LIN {X 0,Y 334.932,Z 502.73,A -85,B 0,C 180,E1 -14665.187,E2 -14665.187} C_VEL
LIN {X 0,Y 334.415,Z 506.51,A -85,B 0,C 180,E1 -14666.99,E2 -14666.99} C_VEL
LIN {X 0,Y 334.012,Z 509.299,A -85,B 0,C 180,E1 -14668.796,E2 -14668.796} C_VEL
LIN {X 0,Y 333.863,Z 511.532,A -85,B 0,C 180,E1 -14671.207,E2 -14671.207} C_VEL
LIN {X 0,Y 333.779,Z 512.102,A -85,B 0,C 180,E1 -14672.415,E2 -14672.415} C_VEL
LIN {X 0,Y 333.646,Z 512.277,A -85,B 0,C 180,E1 -14673.624,E2 -14673.624} C_VEL
LIN {X 0,Y 334.045,Z 511.395,A -85,B 0,C 180,E1 -14676.04,E2 -14676.04} C_VEL
LIN {X 0,Y 334.412,Z 510.379,A -85,B 0,C 180,E1 -14677.245,E2 -14677.245} C_VEL
LIN {X 0,Y 334.959,Z 507.296,A -85,B 0,C 180,E1 -14679.548,E2 -14679.548} C_VEL
LIN {X 0,Y 335.704,Z 503.489,A -85,B 0,C 180,E1 -14681.473,E2 -14681.473} C_VEL
LIN {X 0,Y 336.395,Z 498.792,A -85,B 0,C 180,E1 -14683.287,E2 -14683.287} C_VEL
LIN {X 0,Y 337.32,Z 492.834,A -85,B 0,C 180,E1 -14685.097,E2 -14685.097} C_VEL
LIN {X 0,Y 338.463,Z 485.332,A -85,B 0,C 180,E1 -14686.901,E2 -14686.901} C_VEL
LIN {X 0,Y 339.867,Z 475.902,A -85,B 0,C 180,E1 -14688.695,E2 -14688.695} C_VEL
LIN {X 0,Y 341.064,Z 466.087,A -85,B 0,C 180,E1 -14690.192,E2 -14690.192} C_VEL
LIN {X 0,Y 342.197,Z 454.989,A -85,B 0,C 180,E1 -14691.539,E2 -14691.539} C_VEL
LIN {X 0,Y 343.141,Z 443.458,A -85,B 0,C 180,E1 -14692.639,E2 -14692.639} C_VEL
LIN {X 0,Y 343.723,Z 434.102,A -85,B 0,C 180,E1 -14693.339,E2 -14693.339} C_VEL
LIN {X 0,Y 339.861,Z 422.675,A -85,B 0,C 180,E1 -14694.326,E2 -14694.326} C_VEL
LIN {X 0,Y 334.962,Z 410.747,A -85,B 0,C 180,E1 -14695.19,E2 -14695.19} C_VEL
LIN {X 0,Y 333.811,Z 407.943,A -85,B 0,C 180,E1 -14695.364,E2 -14695.364} C_VEL
LIN {X 0,Y 333.742,Z 407.533,A -85,B 0,C 180,E1 -14695.441,E2 -14695.441} C_VEL
LIN {X 0,Y 333.717,Z 407.543,A -85,B 0,C 180,E1 -14698.973,E2 -14698.973} C_VEL
LIN {X 0,Y 333.649,Z 407.552,A -85,B 0,C 180,E1 -14702.587,E2 -14702.587} C_VEL
LIN {X 0,Y 333.682,Z 407.549,A -85,B 0,C 180,E1 -14706.139,E2 -14706.139} C_VEL
LIN {X 0,Y 333.652,Z 407.539,A -85,B 0,C 180,E1 -14709.193,E2 -14709.193} C_VEL
LIN {X 0,Y 333.638,Z 407.548,A -85,B 0,C 180,E1 -14712.5,E2 -14712.5} C_VEL
LIN {X 0,Y 333.591,Z 407.549,A -85,B 0,C 180,E1 -14716.485,E2 -14716.485} C_VEL
LIN {X 0,Y 333.654,Z 407.539,A -85,B 0,C 180,E1 -14719.315,E2 -14719.315} C_VEL
LIN {X 0,Y 333.642,Z 407.519,A -85,B 0,C 180,E1 -14721.721,E2 -14721.721} C_VEL
LIN {X 0,Y 332.986,Z 407.614,A -85,B 0,C 180,E1 -14722.729,E2 -14722.729} C_VEL
LIN {X 0,Y 330.166,Z 407.982,A -85,B 0,C 180,E1 -14724.369,E2 -14724.369} C_VEL
LIN {X 0,Y 327.763,Z 408.288,A -85,B 0,C 180,E1 -14725.697,E2 -14725.697} C_VEL
LIN {X 0,Y 326.717,Z 408.412,A -85,B 0,C 180,E1 -14726.725,E2 -14726.725} C_VEL
LIN {X 0,Y 326.623,Z 408.419,A -85,B 0,C 180,E1 -14727.073,E2 -14727.073} C_VEL
LIN {X 0,Y 326.653,Z 408.377,A -85,B 0,C 180,E1 -14730.34,E2 -14730.34} C_VEL
LIN {X 0,Y 326.695,Z 408.413,A -85,B 0,C 180,E1 -14734.516,E2 -14734.516} C_VEL
LIN {X 0,Y 326.643,Z 408.545,A -85,B 0,C 180,E1 -14737.811,E2 -14737.811} C_VEL
LIN {X 0,Y 330.893,Z 422.806,A -85,B 0,C 180,E1 -14739.156,E2 -14739.156} C_VEL
LIN {X 0,Y 333.894,Z 433.415,A -85,B 0,C 180,E1 -14740.319,E2 -14740.319} C_VEL
LIN {X 0,Y 332.75,Z 446.544,A -85,B 0,C 180,E1 -14741.759,E2 -14741.759} C_VEL
LIN {X 0,Y 331.562,Z 458.658,A -85,B 0,C 180,E1 -14743.372,E2 -14743.372} C_VEL
LIN {X 0,Y 330.264,Z 470.023,A -85,B 0,C 180,E1 -14745.205,E2 -14745.205} C_VEL
LIN {X 0,Y 329.393,Z 479.499,A -85,B 0,C 180,E1 -14747.054,E2 -14747.054} C_VEL
LIN {X 0,Y 328.405,Z 488.672,A -85,B 0,C 180,E1 -14749.207,E2 -14749.207} C_VEL
LIN {X 0,Y 327.734,Z 496.151,A -85,B 0,C 180,E1 -14751.366,E2 -14751.366} C_VEL
LIN {X 0,Y 327.381,Z 501.397,A -85,B 0,C 180,E1 -14753.219,E2 -14753.219} C_VEL
LIN {X 0,Y 326.834,Z 505.753,A -85,B 0,C 180,E1 -14755.065,E2 -14755.065} C_VEL
LIN {X 0,Y 326.643,Z 508.141,A -85,B 0,C 180,E1 -14756.299,E2 -14756.299} C_VEL
LIN {X 0,Y 326.854,Z 511.779,A -85,B 0,C 180,E1 -14758.768,E2 -14758.768} C_VEL
LIN {X 0,Y 326.937,Z 514.089,A -85,B 0,C 180,E1 -14761.231,E2 -14761.231} C_VEL
LIN {X 0,Y 327.345,Z 515.047,A -85,B 0,C 180,E1 -14763.693,E2 -14763.693} C_VEL
LIN {X 0,Y 327.978,Z 514.689,A -85,B 0,C 180,E1 -14766.15,E2 -14766.15} C_VEL
LIN {X 0,Y 328.936,Z 512.991,A -85,B 0,C 180,E1 -14768.601,E2 -14768.601} C_VEL
LIN {X 0,Y 330.253,Z 509.9,A -85,B 0,C 180,E1 -14771.042,E2 -14771.042} C_VEL
LIN {X 0,Y 331.845,Z 505.402,A -85,B 0,C 180,E1 -14773.471,E2 -14773.471} C_VEL
LIN {X 0,Y 333.337,Z 501.026,A -85,B 0,C 180,E1 -14775.28,E2 -14775.28} C_VEL
LIN {X 0,Y 335.699,Z 493.646,A -85,B 0,C 180,E1 -14777.672,E2 -14777.672} C_VEL
LIN {X 0,Y 338.143,Z 485.587,A -85,B 0,C 180,E1 -14779.739,E2 -14779.739} C_VEL
LIN {X 0,Y 340.863,Z 475.682,A -85,B 0,C 180,E1 -14781.785,E2 -14781.785} C_VEL
LIN {X 0,Y 343.444,Z 465.427,A -85,B 0,C 180,E1 -14783.518,E2 -14783.518} C_VEL
LIN {X 0,Y 346.007,Z 454.2,A -85,B 0,C 180,E1 -14785.088,E2 -14785.088} C_VEL
LIN {X 0,Y 346.695,Z 451.167,A -85,B 0,C 180,E1 -14785.448,E2 -14785.448} C_VEL
LIN {X 0,Y 346.751,Z 449.531,A -85,B 0,C 180,E1 -14785.698,E2 -14785.698} C_VEL
LIN {X 0,Y 344.955,Z 442.595,A -85,B 0,C 180,E1 -14787.072,E2 -14787.072} C_VEL
LIN {X 0,Y 342.423,Z 435.536,A -85,B 0,C 180,E1 -14788.594,E2 -14788.594} C_VEL
LIN {X 0,Y 338.778,Z 427.656,A -85,B 0,C 180,E1 -14790.489,E2 -14790.489} C_VEL
LIN {X 0,Y 336.804,Z 424.314,A -85,B 0,C 180,E1 -14791.444,E2 -14791.444} C_VEL
LIN {X 0,Y 334.026,Z 421.028,A -85,B 0,C 180,E1 -14792.688,E2 -14792.688} C_VEL
LIN {X 0,Y 331.005,Z 418.156,A -85,B 0,C 180,E1 -14794.099,E2 -14794.099} C_VEL
LIN {X 0,Y 328.685,Z 416.422,A -85,B 0,C 180,E1 -14795.262,E2 -14795.262} C_VEL
LIN {X 0,Y 328.179,Z 415.479,A -85,B 0,C 180,E1 -14795.701,E2 -14795.701} C_VEL
LIN {X 0,Y 328.67,Z 417.798,A -85,B 0,C 180,E1 -14798.324,E2 -14798.324} C_VEL
LIN {X 0,Y 329.451,Z 421.54,A -85,B 0,C 180,E1 -14801.699,E2 -14801.699} C_VEL
LIN {X 0,Y 330.309,Z 425.475,A -85,B 0,C 180,E1 -14804.599,E2 -14804.599} C_VEL
LIN {X 0,Y 331.337,Z 430.877,A -85,B 0,C 180,E1 -14807.935,E2 -14807.935} C_VEL
LIN {X 0,Y 331.487,Z 434.338,A -85,B 0,C 180,E1 -14809.752,E2 -14809.752} C_VEL
LIN {X 0,Y 329.383,Z 444.47,A -85,B 0,C 180,E1 -14814.174,E2 -14814.174} C_VEL
LIN {X 0,Y 329.004,Z 447.721,A -85,B 0,C 180,E1 -14815.43,E2 -14815.43} C_VEL
LIN {X 0,Y 330.074,Z 452.747,A -85,B 0,C 180,E1 -14816.199,E2 -14816.199} C_VEL
LIN {X 0,Y 331.177,Z 456.012,A -85,B 0,C 180,E1 -14816.784,E2 -14816.784} C_VEL
LIN {X 0,Y 332.291,Z 460.774,A -85,B 0,C 180,E1 -14817.472,E2 -14817.472} C_VEL
LIN {X 0,Y 333.055,Z 464.005,A -85,B 0,C 180,E1 -14817.942,E2 -14817.942} C_VEL
LIN {X 0,Y 334.284,Z 469.371,A -85,B 0,C 180,E1 -14818.683,E2 -14818.683} C_VEL
LIN {X 0,Y 336.767,Z 483.631,A -85,B 0,C 180,E1 -14820.487,E2 -14820.487} C_VEL
LIN {X 0,Y 338.023,Z 497.366,A -85,B 0,C 180,E1 -14822.075,E2 -14822.075} C_VEL
LIN {X 0,Y 338.104,Z 510.892,A -85,B 0,C 180,E1 -14823.59,E2 -14823.59} C_VEL
LIN {X 0,Y 336.94,Z 523.468,A -85,B 0,C 180,E1 -14825.014,E2 -14825.014} C_VEL
LIN {X 0,Y 335.439,Z 536.699,A -85,B 0,C 180,E1 -14826.704,E2 -14826.704} C_VEL
LIN {X 0,Y 332.995,Z 548.466,A -85,B 0,C 180,E1 -14828.356,E2 -14828.356} C_VEL
LIN {X 0,Y 330.787,Z 559.176,A -85,B 0,C 180,E1 -14830.126,E2 -14830.126} C_VEL
LIN {X 0,Y 328.676,Z 570.047,A -85,B 0,C 180,E1 -14832.258,E2 -14832.258} C_VEL
LIN {X 0,Y 327.218,Z 579.19,A -85,B 0,C 180,E1 -14834.425,E2 -14834.425} C_VEL
LIN {X 0,Y 326.321,Z 585.851,A -85,B 0,C 180,E1 -14836.295,E2 -14836.295} C_VEL
LIN {X 0,Y 325.733,Z 593.228,A -85,B 0,C 180,E1 -14838.802,E2 -14838.802} C_VEL
LIN {X 0,Y 325.614,Z 598.959,A -85,B 0,C 180,E1 -14841.309,E2 -14841.309} C_VEL
LIN {X 0,Y 325.829,Z 603.168,A -85,B 0,C 180,E1 -14843.807,E2 -14843.807} C_VEL
LIN {X 0,Y 326.041,Z 604.717,A -85,B 0,C 180,E1 -14845.052,E2 -14845.052} C_VEL
LIN {X 0,Y 326.172,Z 605.881,A -85,B 0,C 180,E1 -14846.292,E2 -14846.292} C_VEL
LIN {X 0,Y 326.574,Z 607.099,A -85,B 0,C 180,E1 -14848.766,E2 -14848.766} C_VEL
LIN {X 0,Y 326.764,Z 607.138,A -85,B 0,C 180,E1 -14849.999,E2 -14849.999} C_VEL
LIN {X 0,Y 326.616,Z 606.741,A -85,B 0,C 180,E1 -14851.232,E2 -14851.232} C_VEL
LIN {X 0,Y 326.459,Z 605.959,A -85,B 0,C 180,E1 -14852.466,E2 -14852.466} C_VEL
LIN {X 0,Y 326.23,Z 603.225,A -85,B 0,C 180,E1 -14854.942,E2 -14854.942} C_VEL
LIN {X 0,Y 326.053,Z 599.629,A -85,B 0,C 180,E1 -14857.027,E2 -14857.027} C_VEL
LIN {X 0,Y 325.922,Z 594.313,A -85,B 0,C 180,E1 -14859.306,E2 -14859.306} C_VEL
LIN {X 0,Y 326.074,Z 587.723,A -85,B 0,C 180,E1 -14861.499,E2 -14861.499} C_VEL
LIN {X 0,Y 326.518,Z 579.433,A -85,B 0,C 180,E1 -14863.694,E2 -14863.694} C_VEL
LIN {X 0,Y 327.31,Z 570.812,A -85,B 0,C 180,E1 -14865.568,E2 -14865.568} C_VEL
LIN {X 0,Y 328.372,Z 560.421,A -85,B 0,C 180,E1 -14867.434,E2 -14867.434} C_VEL
LIN {X 0,Y 329.62,Z 550.112,A -85,B 0,C 180,E1 -14868.973,E2 -14868.973} C_VEL
LIN {X 0,Y 331.041,Z 537.717,A -85,B 0,C 180,E1 -14870.504,E2 -14870.504} C_VEL
LIN {X 0,Y 331.642,Z 529.973,A -85,B 0,C 180,E1 -14871.322,E2 -14871.322} C_VEL
LIN {X 0,Y 330.688,Z 516.048,A -85,B 0,C 180,E1 -14872.603,E2 -14872.603} C_VEL
LIN {X 0,Y 329.222,Z 500.525,A -85,B 0,C 180,E1 -14873.76,E2 -14873.76} C_VEL
LIN {X 0,Y 327.764,Z 485.333,A -85,B 0,C 180,E1 -14874.63,E2 -14874.63} C_VEL
LIN {X 0,Y 326.846,Z 476.144,A -85,B 0,C 180,E1 -14875.043,E2 -14875.043} C_VEL
LIN {X 0,Y 327.719,Z 465.495,A -85,B 0,C 180,E1 -14878.914,E2 -14878.914} C_VEL
LIN {X 0,Y 328.904,Z 454.506,A -85,B 0,C 180,E1 -14882.961,E2 -14882.961} C_VEL
LIN {X 0,Y 330.094,Z 444.79,A -85,B 0,C 180,E1 -14886.592,E2 -14886.592} C_VEL
LIN {X 0,Y 331.502,Z 435.163,A -85,B 0,C 180,E1 -14890.251,E2 -14890.251} C_VEL
LIN {X 0,Y 331.337,Z 431.895,A -85,B 0,C 180,E1 -14891.564,E2 -14891.564} C_VEL
LIN {X 0,Y 329.548,Z 423.114,A -85,B 0,C 180,E1 -14895.27,E2 -14895.27} C_VEL
LIN {X 0,Y 327.775,Z 414.147,A -85,B 0,C 180,E1 -14899.251,E2 -14899.251} C_VEL
LIN {X 0,Y 326.642,Z 408.424,A -85,B 0,C 180,E1 -14901.952,E2 -14901.952} C_VEL
LIN {X 0,Y 326.598,Z 408.425,A -85,B 0,C 180,E1 -14905.98,E2 -14905.98} C_VEL
LIN {X 0,Y 326.651,Z 408.417,A -85,B 0,C 180,E1 -14910.34,E2 -14910.34} C_VEL
LIN {X 0,Y 326.68,Z 408.415,A -85,B 0,C 180,E1 -14914.516,E2 -14914.516} C_VEL
LIN {X 0,Y 326.636,Z 408.421,A -85,B 0,C 180,E1 -14918.545,E2 -14918.545} C_VEL
LIN {X 0,Y 326.734,Z 408.412,A -85,B 0,C 180,E1 -14921.177,E2 -14921.177} C_VEL
LIN {X 0,Y 326.753,Z 408.407,A -85,B 0,C 180,E1 -14925.433,E2 -14925.433} C_VEL
LIN {X 0,Y 326.763,Z 408.408,A -85,B 0,C 180,E1 -14928.839,E2 -14928.839} C_VEL
LIN {X 0,Y 326.969,Z 408.381,A -85,B 0,C 180,E1 -14932.59,E2 -14932.59} C_VEL
LIN {X 0,Y 326.77,Z 408.406,A -85,B 0,C 180,E1 -14935.065,E2 -14935.065} C_VEL
LIN {X 0,Y 327.059,Z 408.368,A -85,B 0,C 180,E1 -14937.537,E2 -14937.537} C_VEL
LIN {X 0,Y 327.208,Z 408.348,A -85,B 0,C 180,E1 -14940,E2 -14940} C_VEL
LIN {X 0,Y 327.059,Z 408.369,A -85,B 0,C 180,E1 -14942.463,E2 -14942.463} C_VEL
LIN {X 0,Y 326.961,Z 408.375,A -85,B 0,C 180,E1 -14946.673,E2 -14946.673} C_VEL
LIN {X 0,Y 326.806,Z 408.393,A -85,B 0,C 180,E1 -14949.907,E2 -14949.907} C_VEL
LIN {X 0,Y 326.751,Z 408.406,A -85,B 0,C 180,E1 -14953.686,E2 -14953.686} C_VEL
LIN {X 0,Y 326.69,Z 408.412,A -85,B 0,C 180,E1 -14957.529,E2 -14957.529} C_VEL
LIN {X 0,Y 326.656,Z 408.418,A -85,B 0,C 180,E1 -14960.136,E2 -14960.136} C_VEL
LIN {X 0,Y 326.643,Z 408.42,A -85,B 0,C 180,E1 -14964.13,E2 -14964.13} C_VEL
LIN {X 0,Y 326.677,Z 408.416,A -85,B 0,C 180,E1 -14966.859,E2 -14966.859} C_VEL
LIN {X 0,Y 326.631,Z 408.418,A -85,B 0,C 180,E1 -14970.612,E2 -14970.612} C_VEL
LIN {X 0,Y 326.6,Z 408.425,A -85,B 0,C 180,E1 -14974.021,E2 -14974.021} C_VEL
LIN {X 0,Y 326.622,Z 408.418,A -85,B 0,C 180,E1 -14977.24,E2 -14977.24} C_VEL
LIN {X 0,Y 326.572,Z 408.429,A -85,B 0,C 180,E1 -14981.133,E2 -14981.133} C_VEL
LIN {X 0,Y 326.555,Z 408.43,A -85,B 0,C 180,E1 -14984.75,E2 -14984.75} C_VEL
LIN {X 0,Y 326.594,Z 408.428,A -85,B 0,C 180,E1 -14988.159,E2 -14988.159} C_VEL
LIN {X 0,Y 326.641,Z 408.418,A -85,B 0,C 180,E1 -14991.396,E2 -14991.396} C_VEL
LIN {X 0,Y 326.618,Z 408.424,A -85,B 0,C 180,E1 -14994.853,E2 -14994.853} C_VEL
LIN {X 0,Y 326.608,Z 408.423,A -85,B 0,C 180,E1 -14997.458,E2 -14997.458} C_VEL
LIN {X 0,Y 326.659,Z 408.421,A -85,B 0,C 180,E1 -15000.343,E2 -15000.343} C_VEL
LIN {X 0,Y 326.689,Z 408.417,A -85,B 0,C 180,E1 -15004.518,E2 -15004.518} C_VEL
LIN {X 0,Y 326.649,Z 408.424,A -85,B 0,C 180,E1 -15008.547,E2 -15008.547} C_VEL
LIN {X 0,Y 326.765,Z 408.401,A -85,B 0,C 180,E1 -15011.359,E2 -15011.359} C_VEL
LIN {X 0,Y 329.107,Z 414.783,A -85,B 0,C 180,E1 -15011.735,E2 -15011.735} C_VEL
LIN {X 0,Y 333.389,Z 426.874,A -85,B 0,C 180,E1 -15012.597,E2 -15012.597} C_VEL
LIN {X 0,Y 335.235,Z 432.94,A -85,B 0,C 180,E1 -15013.099,E2 -15013.099} C_VEL
LIN {X 0,Y 334.504,Z 445.35,A -85,B 0,C 180,E1 -15014.037,E2 -15014.037} C_VEL
LIN {X 0,Y 333.612,Z 457.021,A -85,B 0,C 180,E1 -15015.202,E2 -15015.202} C_VEL
LIN {X 0,Y 332.529,Z 467.779,A -85,B 0,C 180,E1 -15016.558,E2 -15016.558} C_VEL
LIN {X 0,Y 331.382,Z 477.329,A -85,B 0,C 180,E1 -15018.068,E2 -15018.068} C_VEL
LIN {X 0,Y 330.415,Z 485.149,A -85,B 0,C 180,E1 -15019.585,E2 -15019.585} C_VEL
LIN {X 0,Y 329.304,Z 492.836,A -85,B 0,C 180,E1 -15021.41,E2 -15021.41} C_VEL
LIN {X 0,Y 328.566,Z 498.963,A -85,B 0,C 180,E1 -15023.245,E2 -15023.245} C_VEL
LIN {X 0,Y 327.945,Z 503.816,A -85,B 0,C 180,E1 -15025.084,E2 -15025.084} C_VEL
LIN {X 0,Y 327.404,Z 507.577,A -85,B 0,C 180,E1 -15026.925,E2 -15026.925} C_VEL
LIN {X 0,Y 326.989,Z 510.346,A -85,B 0,C 180,E1 -15028.77,E2 -15028.77} C_VEL
LIN {X 0,Y 326.846,Z 512.559,A -85,B 0,C 180,E1 -15031.233,E2 -15031.233} C_VEL
LIN {X 0,Y 326.754,Z 513.12,A -85,B 0,C 180,E1 -15032.467,E2 -15032.467} C_VEL
LIN {X 0,Y 326.623,Z 513.277,A -85,B 0,C 180,E1 -15033.702,E2 -15033.702} C_VEL
LIN {X 0,Y 327.051,Z 512.375,A -85,B 0,C 180,E1 -15036.169,E2 -15036.169} C_VEL
LIN {X 0,Y 327.436,Z 511.345,A -85,B 0,C 180,E1 -15037.4,E2 -15037.4} C_VEL
LIN {X 0,Y 327.99,Z 508.307,A -85,B 0,C 180,E1 -15039.71,E2 -15039.71} C_VEL
LIN {X 0,Y 328.79,Z 504.409,A -85,B 0,C 180,E1 -15041.718,E2 -15041.718} C_VEL
LIN {X 0,Y 329.535,Z 499.688,A -85,B 0,C 180,E1 -15043.569,E2 -15043.569} C_VEL
LIN {X 0,Y 330.517,Z 493.703,A -85,B 0,C 180,E1 -15045.415,E2 -15045.415} C_VEL
LIN {X 0,Y 331.731,Z 486.153,A -85,B 0,C 180,E1 -15047.255,E2 -15047.255} C_VEL
LIN {X 0,Y 333.199,Z 476.686,A -85,B 0,C 180,E1 -15049.084,E2 -15049.084} C_VEL
LIN {X 0,Y 334.456,Z 466.801,A -85,B 0,C 180,E1 -15050.609,E2 -15050.609} C_VEL
LIN {X 0,Y 335.623,Z 455.641,A -85,B 0,C 180,E1 -15051.983,E2 -15051.983} C_VEL
LIN {X 0,Y 336.557,Z 444.782,A -85,B 0,C 180,E1 -15053.037,E2 -15053.037} C_VEL
LIN {X 0,Y 337.171,Z 436.006,A -85,B 0,C 180,E1 -15053.709,E2 -15053.709} C_VEL
LIN {X 0,Y 333.326,Z 424.538,A -85,B 0,C 180,E1 -15054.749,E2 -15054.749} C_VEL
LIN {X 0,Y 328.591,Z 413.222,A -85,B 0,C 180,E1 -15055.623,E2 -15055.623} C_VEL
LIN {X 0,Y 326.744,Z 408.688,A -85,B 0,C 180,E1 -15055.913,E2 -15055.913} C_VEL
LIN {X 0,Y 326.71,Z 408.413,A -85,B 0,C 180,E1 -15056.037,E2 -15056.037} C_VEL
LIN {X 0,Y 326.666,Z 408.421,A -85,B 0,C 180,E1 -15059.66,E2 -15059.66} C_VEL
LIN {X 0,Y 326.613,Z 408.43,A -85,B 0,C 180,E1 -15064.02,E2 -15064.02} C_VEL
LIN {X 0,Y 326.633,Z 408.415,A -85,B 0,C 180,E1 -15067.239,E2 -15067.239} C_VEL
LIN {X 0,Y 326.583,Z 408.429,A -85,B 0,C 180,E1 -15071.132,E2 -15071.132} C_VEL
LIN {X 0,Y 326.535,Z 408.432,A -85,B 0,C 180,E1 -15074.743,E2 -15074.743} C_VEL
LIN {X 0,Y 326.584,Z 408.428,A -85,B 0,C 180,E1 -15078.155,E2 -15078.155} C_VEL
LIN {X 0,Y 326.594,Z 408.396,A -85,B 0,C 180,E1 -15081.718,E2 -15081.718} C_VEL
LIN {X 0,Y 326.625,Z 408.423,A -85,B 0,C 180,E1 -15084.851,E2 -15084.851} C_VEL
LIN {X 0,Y 326.623,Z 408.419,A -85,B 0,C 180,E1 -15087.073,E2 -15087.073} C_VEL
LIN {X 0,Y 325.945,Z 408.491,A -85,B 0,C 180,E1 -15088.101,E2 -15088.101} C_VEL
LIN {X 0,Y 323.129,Z 408.834,A -85,B 0,C 180,E1 -15089.776,E2 -15089.776} C_VEL
LIN {X 0,Y 320.743,Z 409.13,A -85,B 0,C 180,E1 -15091.132,E2 -15091.132} C_VEL
LIN {X 0,Y 319.703,Z 409.262,A -85,B 0,C 180,E1 -15092.181,E2 -15092.181} C_VEL
LIN {X 0,Y 319.609,Z 409.275,A -85,B 0,C 180,E1 -15092.537,E2 -15092.537} C_VEL
LIN {X 0,Y 319.608,Z 409.298,A -85,B 0,C 180,E1 -15095.304,E2 -15095.304} C_VEL
LIN {X 0,Y 319.601,Z 409.359,A -85,B 0,C 180,E1 -15097.487,E2 -15097.487} C_VEL
LIN {X 0,Y 323.434,Z 422.34,A -85,B 0,C 180,E1 -15098.718,E2 -15098.718} C_VEL
LIN {X 0,Y 326.81,Z 434.237,A -85,B 0,C 180,E1 -15100.038,E2 -15100.038} C_VEL
LIN {X 0,Y 326.804,Z 437.302,A -85,B 0,C 180,E1 -15100.365,E2 -15100.365} C_VEL
LIN {X 0,Y 325.561,Z 450.343,A -85,B 0,C 180,E1 -15101.89,E2 -15101.89} C_VEL
LIN {X 0,Y 324.224,Z 462.54,A -85,B 0,C 180,E1 -15103.632,E2 -15103.632} C_VEL
LIN {X 0,Y 323.024,Z 473.423,A -85,B 0,C 180,E1 -15105.51,E2 -15105.51} C_VEL
LIN {X 0,Y 322.138,Z 482.533,A -85,B 0,C 180,E1 -15107.398,E2 -15107.398} C_VEL
LIN {X 0,Y 321.239,Z 491.376,A -85,B 0,C 180,E1 -15109.601,E2 -15109.601} C_VEL
LIN {X 0,Y 320.63,Z 498.558,A -85,B 0,C 180,E1 -15111.809,E2 -15111.809} C_VEL
LIN {X 0,Y 320.185,Z 503.615,A -85,B 0,C 180,E1 -15113.699,E2 -15113.699} C_VEL
LIN {X 0,Y 319.604,Z 508.942,A -85,B 0,C 180,E1 -15116.217,E2 -15116.217} C_VEL
LIN {X 0,Y 319.836,Z 512.709,A -85,B 0,C 180,E1 -15118.741,E2 -15118.741} C_VEL
LIN {X 0,Y 319.918,Z 515.143,A -85,B 0,C 180,E1 -15121.258,E2 -15121.258} C_VEL
LIN {X 0,Y 320.356,Z 516.234,A -85,B 0,C 180,E1 -15123.773,E2 -15123.773} C_VEL
LIN {X 0,Y 321.05,Z 516.007,A -85,B 0,C 180,E1 -15126.284,E2 -15126.284} C_VEL
LIN {X 0,Y 322.073,Z 514.47,A -85,B 0,C 180,E1 -15128.786,E2 -15128.786} C_VEL
LIN {X 0,Y 323.495,Z 511.557,A -85,B 0,C 180,E1 -15131.275,E2 -15131.275} C_VEL
LIN {X 0,Y 325.18,Z 507.234,A -85,B 0,C 180,E1 -15133.753,E2 -15133.753} C_VEL
LIN {X 0,Y 327.371,Z 501.372,A -85,B 0,C 180,E1 -15136.205,E2 -15136.205} C_VEL
LIN {X 0,Y 329.628,Z 494.853,A -85,B 0,C 180,E1 -15138.329,E2 -15138.329} C_VEL
LIN {X 0,Y 332.263,Z 486.832,A -85,B 0,C 180,E1 -15140.426,E2 -15140.426} C_VEL
LIN {X 0,Y 335.178,Z 476.997,A -85,B 0,C 180,E1 -15142.496,E2 -15142.496} C_VEL
LIN {X 0,Y 337.936,Z 466.841,A -85,B 0,C 180,E1 -15144.251,E2 -15144.251} C_VEL
LIN {X 0,Y 340.876,Z 455.089,A -85,B 0,C 180,E1 -15145.915,E2 -15145.915} C_VEL
LIN {X 0,Y 341.255,Z 453.273,A -85,B 0,C 180,E1 -15146.143,E2 -15146.143} C_VEL
LIN {X 0,Y 339.689,Z 446.272,A -85,B 0,C 180,E1 -15147.623,E2 -15147.623} C_VEL
LIN {X 0,Y 337.165,Z 438.886,A -85,B 0,C 180,E1 -15149.331,E2 -15149.331} C_VEL
LIN {X 0,Y 334.214,Z 432.295,A -85,B 0,C 180,E1 -15151.081,E2 -15151.081} C_VEL
LIN {X 0,Y 332.185,Z 428.884,A -85,B 0,C 180,E1 -15152.19,E2 -15152.19} C_VEL
LIN {X 0,Y 329.068,Z 425.661,A -85,B 0,C 180,E1 -15153.73,E2 -15153.73} C_VEL
LIN {X 0,Y 325.683,Z 422.478,A -85,B 0,C 180,E1 -15155.636,E2 -15155.636} C_VEL
LIN {X 0,Y 322.565,Z 420.962,A -85,B 0,C 180,E1 -15157.594,E2 -15157.594} C_VEL
LIN {X 0,Y 321.917,Z 419.977,A -85,B 0,C 180,E1 -15158.286,E2 -15158.286} C_VEL
LIN {X 0,Y 322.479,Z 422.688,A -85,B 0,C 180,E1 -15160.829,E2 -15160.829} C_VEL
LIN {X 0,Y 323.398,Z 426.99,A -85,B 0,C 180,E1 -15164.179,E2 -15164.179} C_VEL
LIN {X 0,Y 324.372,Z 432.056,A -85,B 0,C 180,E1 -15167.447,E2 -15167.447} C_VEL
LIN {X 0,Y 324.643,Z 435.778,A -85,B 0,C 180,E1 -15169.499,E2 -15169.499} C_VEL
LIN {X 0,Y 322.913,Z 443.641,A -85,B 0,C 180,E1 -15173.004,E2 -15173.004} C_VEL
LIN {X 0,Y 323.599,Z 447.88,A -85,B 0,C 180,E1 -15173.766,E2 -15173.766} C_VEL
LIN {X 0,Y 325.045,Z 452.168,A -85,B 0,C 180,E1 -15174.728,E2 -15174.728} C_VEL
LIN {X 0,Y 326.063,Z 457.387,A -85,B 0,C 180,E1 -15175.584,E2 -15175.584} C_VEL
LIN {X 0,Y 326.953,Z 460.883,A -85,B 0,C 180,E1 -15176.206,E2 -15176.206} C_VEL
LIN {X 0,Y 328.451,Z 468.009,A -85,B 0,C 180,E1 -15177.314,E2 -15177.314} C_VEL
LIN {X 0,Y 330.24,Z 478.17,A -85,B 0,C 180,E1 -15178.769,E2 -15178.769} C_VEL
LIN {X 0,Y 331.683,Z 490.05,A -85,B 0,C 180,E1 -15180.313,E2 -15180.313} C_VEL
LIN {X 0,Y 332.228,Z 502.351,A -85,B 0,C 180,E1 -15181.81,E2 -15181.81} C_VEL
LIN {X 0,Y 331.93,Z 513.787,A -85,B 0,C 180,E1 -15183.182,E2 -15183.182} C_VEL
LIN {X 0,Y 330.138,Z 528.402,A -85,B 0,C 180,E1 -15184.968,E2 -15184.968} C_VEL
LIN {X 0,Y 328.408,Z 540.637,A -85,B 0,C 180,E1 -15186.676,E2 -15186.676} C_VEL
LIN {X 0,Y 325.584,Z 552.334,A -85,B 0,C 180,E1 -15188.471,E2 -15188.471} C_VEL
LIN {X 0,Y 323.096,Z 563.972,A -85,B 0,C 180,E1 -15190.626,E2 -15190.626} C_VEL
LIN {X 0,Y 321.1,Z 573.791,A -85,B 0,C 180,E1 -15192.813,E2 -15192.813} C_VEL
LIN {X 0,Y 319.774,Z 582.115,A -85,B 0,C 180,E1 -15195.04,E2 -15195.04} C_VEL
LIN {X 0,Y 318.933,Z 589.04,A -85,B 0,C 180,E1 -15197.269,E2 -15197.269} C_VEL
LIN {X 0,Y 318.543,Z 595.438,A -85,B 0,C 180,E1 -15199.833,E2 -15199.833} C_VEL
LIN {X 0,Y 318.624,Z 600.306,A -85,B 0,C 180,E1 -15202.394,E2 -15202.394} C_VEL
LIN {X 0,Y 318.974,Z 603.685,A -85,B 0,C 180,E1 -15204.943,E2 -15204.943} C_VEL
LIN {X 0,Y 319.12,Z 604.813,A -85,B 0,C 180,E1 -15206.21,E2 -15206.21} C_VEL
LIN {X 0,Y 319.566,Z 605.957,A -85,B 0,C 180,E1 -15208.738,E2 -15208.738} C_VEL
LIN {X 0,Y 319.757,Z 605.958,A -85,B 0,C 180,E1 -15209.999,E2 -15209.999} C_VEL
LIN {X 0,Y 319.613,Z 605.524,A -85,B 0,C 180,E1 -15211.259,E2 -15211.259} C_VEL
LIN {X 0,Y 319.455,Z 604.697,A -85,B 0,C 180,E1 -15212.52,E2 -15212.52} C_VEL
LIN {X 0,Y 319.203,Z 601.857,A -85,B 0,C 180,E1 -15215.051,E2 -15215.051} C_VEL
LIN {X 0,Y 319.034,Z 598.3,A -85,B 0,C 180,E1 -15217.116,E2 -15217.116} C_VEL
LIN {X 0,Y 318.909,Z 592.743,A -85,B 0,C 180,E1 -15219.512,E2 -15219.512} C_VEL
LIN {X 0,Y 319.061,Z 585.993,A -85,B 0,C 180,E1 -15221.755,E2 -15221.755} C_VEL
LIN {X 0,Y 319.562,Z 577.558,A -85,B 0,C 180,E1 -15223.998,E2 -15223.998} C_VEL
LIN {X 0,Y 320.388,Z 568.787,A -85,B 0,C 180,E1 -15225.913,E2 -15225.913} C_VEL
LIN {X 0,Y 321.559,Z 558.236,A -85,B 0,C 180,E1 -15227.816,E2 -15227.816} C_VEL
LIN {X 0,Y 322.928,Z 546.566,A -85,B 0,C 180,E1 -15229.547,E2 -15229.547} C_VEL
LIN {X 0,Y 324.269,Z 535.355,A -85,B 0,C 180,E1 -15230.915,E2 -15230.915} C_VEL
LIN {X 0,Y 324.609,Z 530.712,A -85,B 0,C 180,E1 -15231.412,E2 -15231.412} C_VEL
LIN {X 0,Y 323.724,Z 517.023,A -85,B 0,C 180,E1 -15232.748,E2 -15232.748} C_VEL
LIN {X 0,Y 322.435,Z 502.933,A -85,B 0,C 180,E1 -15233.867,E2 -15233.867} C_VEL
LIN {X 0,Y 320.938,Z 486.828,A -85,B 0,C 180,E1 -15234.86,E2 -15234.86} C_VEL
LIN {X 0,Y 319.82,Z 475.233,A -85,B 0,C 180,E1 -15235.429,E2 -15235.429} C_VEL
LIN {X 0,Y 320.783,Z 464.247,A -85,B 0,C 180,E1 -15239.533,E2 -15239.533} C_VEL
LIN {X 0,Y 322.011,Z 453.616,A -85,B 0,C 180,E1 -15243.545,E2 -15243.545} C_VEL
LIN {X 0,Y 323.126,Z 444.94,A -85,B 0,C 180,E1 -15246.879,E2 -15246.879} C_VEL
LIN {X 0,Y 324.286,Z 437.561,A -85,B 0,C 180,E1 -15249.74,E2 -15249.74} C_VEL
LIN {X 0,Y 324.522,Z 435.11,A -85,B 0,C 180,E1 -15250.714,E2 -15250.714} C_VEL
LIN {X 0,Y 323.913,Z 430.917,A -85,B 0,C 180,E1 -15252.464,E2 -15252.464} C_VEL
LIN {X 0,Y 322.265,Z 422.73,A -85,B 0,C 180,E1 -15256.024,E2 -15256.024} C_VEL
LIN {X 0,Y 320.687,Z 414.845,A -85,B 0,C 180,E1 -15259.619,E2 -15259.619} C_VEL
LIN {X 0,Y 319.605,Z 409.299,A -85,B 0,C 180,E1 -15262.335,E2 -15262.335} C_VEL
LIN {X 0,Y 319.552,Z 409.308,A -85,B 0,C 180,E1 -15265.123,E2 -15265.123} C_VEL
LIN {X 0,Y 319.561,Z 409.306,A -85,B 0,C 180,E1 -15269.057,E2 -15269.057} C_VEL
LIN {X 0,Y 319.599,Z 409.297,A -85,B 0,C 180,E1 -15272.498,E2 -15272.498} C_VEL
LIN {X 0,Y 319.595,Z 409.3,A -85,B 0,C 180,E1 -15275.303,E2 -15275.303} C_VEL
LIN {X 0,Y 319.587,Z 409.298,A -85,B 0,C 180,E1 -15278.047,E2 -15278.047} C_VEL
LIN {X 0,Y 319.679,Z 409.29,A -85,B 0,C 180,E1 -15280.962,E2 -15280.962} C_VEL
LIN {X 0,Y 319.721,Z 409.284,A -85,B 0,C 180,E1 -15285.276,E2 -15285.276} C_VEL
LIN {X 0,Y 319.749,Z 409.275,A -85,B 0,C 180,E1 -15289.873,E2 -15289.873} C_VEL
LIN {X 0,Y 319.923,Z 409.257,A -85,B 0,C 180,E1 -15292.426,E2 -15292.426} C_VEL
LIN {X 0,Y 319.74,Z 409.282,A -85,B 0,C 180,E1 -15294.956,E2 -15294.956} C_VEL
LIN {X 0,Y 319.999,Z 409.248,A -85,B 0,C 180,E1 -15297.483,E2 -15297.483} C_VEL
LIN {X 0,Y 320.159,Z 409.226,A -85,B 0,C 180,E1 -15300,E2 -15300} C_VEL
LIN {X 0,Y 319.999,Z 409.248,A -85,B 0,C 180,E1 -15302.518,E2 -15302.518} C_VEL
LIN {X 0,Y 319.921,Z 409.252,A -85,B 0,C 180,E1 -15306.664,E2 -15306.664} C_VEL
LIN {X 0,Y 319.75,Z 409.271,A -85,B 0,C 180,E1 -15310.128,E2 -15310.128} C_VEL
LIN {X 0,Y 319.721,Z 409.287,A -85,B 0,C 180,E1 -15314.725,E2 -15314.725} C_VEL
LIN {X 0,Y 319.68,Z 409.289,A -85,B 0,C 180,E1 -15319.039,E2 -15319.039} C_VEL
LIN {X 0,Y 319.561,Z 409.302,A -85,B 0,C 180,E1 -15323.321,E2 -15323.321} C_VEL
LIN {X 0,Y 319.627,Z 409.294,A -85,B 0,C 180,E1 -15326.089,E2 -15326.089} C_VEL
LIN {X 0,Y 319.581,Z 409.293,A -85,B 0,C 180,E1 -15328.935,E2 -15328.935} C_VEL
LIN {X 0,Y 319.525,Z 409.303,A -85,B 0,C 180,E1 -15331.863,E2 -15331.863} C_VEL
LIN {X 0,Y 319.573,Z 409.298,A -85,B 0,C 180,E1 -15335.544,E2 -15335.544} C_VEL
LIN {X 0,Y 319.551,Z 409.298,A -85,B 0,C 180,E1 -15338.012,E2 -15338.012} C_VEL
LIN {X 0,Y 319.52,Z 409.306,A -85,B 0,C 180,E1 -15341.599,E2 -15341.599} C_VEL
LIN {X 0,Y 319.54,Z 409.3,A -85,B 0,C 180,E1 -15345.269,E2 -15345.269} C_VEL
LIN {X 0,Y 319.541,Z 409.307,A -85,B 0,C 180,E1 -15348.716,E2 -15348.716} C_VEL
LIN {X 0,Y 319.595,Z 409.3,A -85,B 0,C 180,E1 -15352.341,E2 -15352.341} C_VEL
LIN {X 0,Y 319.558,Z 409.302,A -85,B 0,C 180,E1 -15355.125,E2 -15355.125} C_VEL
LIN {X 0,Y 319.569,Z 409.299,A -85,B 0,C 180,E1 -15359.059,E2 -15359.059} C_VEL
LIN {X 0,Y 319.606,Z 409.299,A -85,B 0,C 180,E1 -15362.5,E2 -15362.5} C_VEL
LIN {X 0,Y 319.605,Z 409.297,A -85,B 0,C 180,E1 -15365.306,E2 -15365.306} C_VEL
LIN {X 0,Y 319.598,Z 409.302,A -85,B 0,C 180,E1 -15368.05,E2 -15368.05} C_VEL
LIN {X 0,Y 319.672,Z 409.285,A -85,B 0,C 180,E1 -15370.896,E2 -15370.896} C_VEL
LIN {X 0,Y 321.437,Z 413.995,A -85,B 0,C 180,E1 -15371.168,E2 -15371.168} C_VEL
LIN {X 0,Y 325.831,Z 425.768,A -85,B 0,C 180,E1 -15372.006,E2 -15372.006} C_VEL
LIN {X 0,Y 328.476,Z 434.433,A -85,B 0,C 180,E1 -15372.734,E2 -15372.734} C_VEL
LIN {X 0,Y 327.776,Z 446.729,A -85,B 0,C 180,E1 -15373.699,E2 -15373.699} C_VEL
LIN {X 0,Y 326.842,Z 458.347,A -85,B 0,C 180,E1 -15374.889,E2 -15374.889} C_VEL
LIN {X 0,Y 325.726,Z 469.027,A -85,B 0,C 180,E1 -15376.272,E2 -15376.272} C_VEL
LIN {X 0,Y 324.54,Z 478.535,A -85,B 0,C 180,E1 -15377.812,E2 -15377.812} C_VEL
LIN {X 0,Y 323.532,Z 486.323,A -85,B 0,C 180,E1 -15379.361,E2 -15379.361} C_VEL
LIN {X 0,Y 322.378,Z 493.981,A -85,B 0,C 180,E1 -15381.224,E2 -15381.224} C_VEL
LIN {X 0,Y 321.622,Z 500.069,A -85,B 0,C 180,E1 -15383.099,E2 -15383.099} C_VEL
LIN {X 0,Y 320.959,Z 504.902,A -85,B 0,C 180,E1 -15384.977,E2 -15384.977} C_VEL
LIN {X 0,Y 320.392,Z 508.643,A -85,B 0,C 180,E1 -15386.858,E2 -15386.858} C_VEL
LIN {X 0,Y 319.966,Z 511.393,A -85,B 0,C 180,E1 -15388.743,E2 -15388.743} C_VEL
LIN {X 0,Y 319.828,Z 513.586,A -85,B 0,C 180,E1 -15391.26,E2 -15391.26} C_VEL
LIN {X 0,Y 319.73,Z 514.136,A -85,B 0,C 180,E1 -15392.521,E2 -15392.521} C_VEL
LIN {X 0,Y 319.602,Z 514.277,A -85,B 0,C 180,E1 -15393.784,E2 -15393.784} C_VEL
LIN {X 0,Y 320.06,Z 513.355,A -85,B 0,C 180,E1 -15396.305,E2 -15396.305} C_VEL
LIN {X 0,Y 320.462,Z 512.309,A -85,B 0,C 180,E1 -15397.562,E2 -15397.562} C_VEL
LIN {X 0,Y 321.033,Z 509.303,A -85,B 0,C 180,E1 -15399.889,E2 -15399.889} C_VEL
LIN {X 0,Y 321.892,Z 505.328,A -85,B 0,C 180,E1 -15401.972,E2 -15401.972} C_VEL
LIN {X 0,Y 322.686,Z 500.583,A -85,B 0,C 180,E1 -15403.863,E2 -15403.863} C_VEL
LIN {X 0,Y 323.726,Z 494.569,A -85,B 0,C 180,E1 -15405.747,E2 -15405.747} C_VEL
LIN {X 0,Y 325.014,Z 486.975,A -85,B 0,C 180,E1 -15407.623,E2 -15407.623} C_VEL
LIN {X 0,Y 326.524,Z 477.475,A -85,B 0,C 180,E1 -15409.49,E2 -15409.49} C_VEL
LIN {X 0,Y 327.867,Z 467.516,A -85,B 0,C 180,E1 -15411.043,E2 -15411.043} C_VEL
LIN {X 0,Y 329.062,Z 456.297,A -85,B 0,C 180,E1 -15412.444,E2 -15412.444} C_VEL
LIN {X 0,Y 330.059,Z 445.319,A -85,B 0,C 180,E1 -15413.517,E2 -15413.517} C_VEL
LIN {X 0,Y 330.585,Z 438.209,A -85,B 0,C 180,E1 -15414.075,E2 -15414.075} C_VEL
LIN {X 0,Y 327.709,Z 429.009,A -85,B 0,C 180,E1 -15414.953,E2 -15414.953} C_VEL
LIN {X 0,Y 323.229,Z 417.688,A -85,B 0,C 180,E1 -15415.905,E2 -15415.905} C_VEL
LIN {X 0,Y 319.791,Z 410.043,A -85,B 0,C 180,E1 -15416.463,E2 -15416.463} C_VEL
LIN {X 0,Y 319.665,Z 409.291,A -85,B 0,C 180,E1 -15416.515,E2 -15416.515} C_VEL
LIN {X 0,Y 319.597,Z 409.303,A -85,B 0,C 180,E1 -15420.384,E2 -15420.384} C_VEL
LIN {X 0,Y 319.582,Z 409.306,A -85,B 0,C 180,E1 -15423.353,E2 -15423.353} C_VEL
LIN {X 0,Y 319.564,Z 409.304,A -85,B 0,C 180,E1 -15426.428,E2 -15426.428} C_VEL
LIN {X 0,Y 319.564,Z 409.298,A -85,B 0,C 180,E1 -15429.669,E2 -15429.669} C_VEL
LIN {X 0,Y 319.528,Z 409.307,A -85,B 0,C 180,E1 -15433.461,E2 -15433.461} C_VEL
LIN {X 0,Y 319.563,Z 409.303,A -85,B 0,C 180,E1 -15437.017,E2 -15437.017} C_VEL
LIN {X 0,Y 319.553,Z 409.276,A -85,B 0,C 180,E1 -15440.371,E2 -15440.371} C_VEL
LIN {X 0,Y 319.586,Z 409.301,A -85,B 0,C 180,E1 -15444.457,E2 -15444.457} C_VEL
LIN {X 0,Y 319.537,Z 409.287,A -85,B 0,C 180,E1 -15448.138,E2 -15448.138} C_VEL
LIN {X 0,Y 319.616,Z 409.261,A -85,B 0,C 180,E1 -15451.59,E2 -15451.59} C_VEL
LIN {X 0,Y 319.609,Z 409.275,A -85,B 0,C 180,E1 -15452.537,E2 -15452.537} C_VEL
LIN {X 0,Y 318.915,Z 409.371,A -85,B 0,C 180,E1 -15453.238,E2 -15453.238} C_VEL
LIN {X 0,Y 316.074,Z 409.737,A -85,B 0,C 180,E1 -15454.336,E2 -15454.336} C_VEL
LIN {X 0,Y 313.222,Z 410.097,A -85,B 0,C 180,E1 -15455.454,E2 -15455.454} C_VEL
LIN {X 0,Y 312.541,Z 410.18,A -85,B 0,C 180,E1 -15456.176,E2 -15456.176} C_VEL
LIN {X 0,Y 312.551,Z 410.178,A -85,B 0,C 180,E1 -15457.158,E2 -15457.158} C_VEL
LIN {X 0,Y 316.453,Z 423.55,A -85,B 0,C 180,E1 -15458.456,E2 -15458.456} C_VEL
LIN {X 0,Y 320.034,Z 436.453,A -85,B 0,C 180,E1 -15459.932,E2 -15459.932} C_VEL
LIN {X 0,Y 318.787,Z 449.444,A -85,B 0,C 180,E1 -15461.44,E2 -15461.44} C_VEL
LIN {X 0,Y 317.515,Z 461.326,A -85,B 0,C 180,E1 -15463.111,E2 -15463.111} C_VEL
LIN {X 0,Y 316.306,Z 471.721,A -85,B 0,C 180,E1 -15464.866,E2 -15464.866} C_VEL
LIN {X 0,Y 315.378,Z 481.254,A -85,B 0,C 180,E1 -15466.796,E2 -15466.796} C_VEL
LIN {X 0,Y 314.352,Z 490.488,A -85,B 0,C 180,E1 -15469.045,E2 -15469.045} C_VEL
LIN {X 0,Y 313.717,Z 497.074,A -85,B 0,C 180,E1 -15470.977,E2 -15470.977} C_VEL
LIN {X 0,Y 313.359,Z 502.597,A -85,B 0,C 180,E1 -15472.914,E2 -15472.914} C_VEL
LIN {X 0,Y 312.726,Z 508.451,A -85,B 0,C 180,E1 -15475.488,E2 -15475.488} C_VEL
LIN {X 0,Y 312.726,Z 511.845,A -85,B 0,C 180,E1 -15477.424,E2 -15477.424} C_VEL
LIN {X 0,Y 312.817,Z 515.081,A -85,B 0,C 180,E1 -15480,E2 -15480} C_VEL
LIN {X 0,Y 313.113,Z 516.973,A -85,B 0,C 180,E1 -15482.573,E2 -15482.573} C_VEL
LIN {X 0,Y 313.692,Z 517.545,A -85,B 0,C 180,E1 -15485.141,E2 -15485.141} C_VEL
LIN {X 0,Y 314.632,Z 516.803,A -85,B 0,C 180,E1 -15487.702,E2 -15487.702} C_VEL
LIN {X 0,Y 315.921,Z 514.754,A -85,B 0,C 180,E1 -15490.251,E2 -15490.251} C_VEL
LIN {X 0,Y 317.619,Z 511.343,A -85,B 0,C 180,E1 -15492.783,E2 -15492.783} C_VEL
LIN {X 0,Y 319.597,Z 506.483,A -85,B 0,C 180,E1 -15495.3,E2 -15495.3} C_VEL
LIN {X 0,Y 322.167,Z 500.016,A -85,B 0,C 180,E1 -15497.782,E2 -15497.782} C_VEL
LIN {X 0,Y 324.817,Z 492.898,A -85,B 0,C 180,E1 -15499.924,E2 -15499.924} C_VEL
LIN {X 0,Y 327.687,Z 484.541,A -85,B 0,C 180,E1 -15501.967,E2 -15501.967} C_VEL
LIN {X 0,Y 330.786,Z 474.387,A -85,B 0,C 180,E1 -15503.992,E2 -15503.992} C_VEL
LIN {X 0,Y 334.145,Z 462.679,A -85,B 0,C 180,E1 -15505.876,E2 -15505.876} C_VEL
LIN {X 0,Y 335.764,Z 455.889,A -85,B 0,C 180,E1 -15506.832,E2 -15506.832} C_VEL
LIN {X 0,Y 333.926,Z 447.859,A -85,B 0,C 180,E1 -15508.691,E2 -15508.691} C_VEL
LIN {X 0,Y 331.054,Z 439.804,A -85,B 0,C 180,E1 -15510.816,E2 -15510.816} C_VEL
LIN {X 0,Y 328.753,Z 435.105,A -85,B 0,C 180,E1 -15512.306,E2 -15512.306} C_VEL
LIN {X 0,Y 327.275,Z 433.285,A -85,B 0,C 180,E1 -15513.122,E2 -15513.122} C_VEL
LIN {X 0,Y 324.609,Z 430.624,A -85,B 0,C 180,E1 -15514.64,E2 -15514.64} C_VEL
LIN {X 0,Y 322.159,Z 428.718,A -85,B 0,C 180,E1 -15516.179,E2 -15516.179} C_VEL
LIN {X 0,Y 319.79,Z 427.18,A -85,B 0,C 180,E1 -15517.977,E2 -15517.977} C_VEL
LIN {X 0,Y 317.58,Z 427.071,A -85,B 0,C 180,E1 -15519.923,E2 -15519.923} C_VEL
LIN {X 0,Y 316.181,Z 427.04,A -85,B 0,C 180,E1 -15522.615,E2 -15522.615} C_VEL
LIN {X 0,Y 317.141,Z 431.634,A -85,B 0,C 180,E1 -15525.911,E2 -15525.911} C_VEL
LIN {X 0,Y 317.818,Z 436.327,A -85,B 0,C 180,E1 -15528.751,E2 -15528.751} C_VEL
LIN {X 0,Y 317.605,Z 438.399,A -85,B 0,C 180,E1 -15529.741,E2 -15529.741} C_VEL
LIN {X 0,Y 318.201,Z 444.051,A -85,B 0,C 180,E1 -15531.068,E2 -15531.068} C_VEL
LIN {X 0,Y 319.446,Z 448.915,A -85,B 0,C 180,E1 -15532.375,E2 -15532.375} C_VEL
LIN {X 0,Y 320.398,Z 454.455,A -85,B 0,C 180,E1 -15533.487,E2 -15533.487} C_VEL
LIN {X 0,Y 321.137,Z 456.936,A -85,B 0,C 180,E1 -15534.07,E2 -15534.07} C_VEL
LIN {X 0,Y 323.362,Z 469.219,A -85,B 0,C 180,E1 -15536.236,E2 -15536.236} C_VEL
LIN {X 0,Y 325.129,Z 481.004,A -85,B 0,C 180,E1 -15538.056,E2 -15538.056} C_VEL
LIN {X 0,Y 326.221,Z 493.315,A -85,B 0,C 180,E1 -15539.764,E2 -15539.764} C_VEL
LIN {X 0,Y 326.384,Z 507.329,A -85,B 0,C 180,E1 -15541.581,E2 -15541.581} C_VEL
LIN {X 0,Y 325.34,Z 520.037,A -85,B 0,C 180,E1 -15543.195,E2 -15543.195} C_VEL
LIN {X 0,Y 322.935,Z 535.147,A -85,B 0,C 180,E1 -15545.231,E2 -15545.231} C_VEL
LIN {X 0,Y 321.947,Z 541.35,A -85,B 0,C 180,E1 -15546.18,E2 -15546.18} C_VEL
LIN {X 0,Y 318.588,Z 554.337,A -85,B 0,C 180,E1 -15548.314,E2 -15548.314} C_VEL
LIN {X 0,Y 316.005,Z 565.368,A -85,B 0,C 180,E1 -15550.511,E2 -15550.511} C_VEL
LIN {X 0,Y 314.011,Z 574.733,A -85,B 0,C 180,E1 -15552.748,E2 -15552.748} C_VEL
LIN {X 0,Y 312.553,Z 583.279,A -85,B 0,C 180,E1 -15555.215,E2 -15555.215} C_VEL
LIN {X 0,Y 311.758,Z 590.105,A -85,B 0,C 180,E1 -15557.632,E2 -15557.632} C_VEL
LIN {X 0,Y 311.445,Z 595.971,A -85,B 0,C 180,E1 -15560.255,E2 -15560.255} C_VEL
LIN {X 0,Y 311.61,Z 600.399,A -85,B 0,C 180,E1 -15562.916,E2 -15562.916} C_VEL
LIN {X 0,Y 311.909,Z 602.663,A -85,B 0,C 180,E1 -15564.828,E2 -15564.828} C_VEL
LIN {X 0,Y 312.067,Z 603.747,A -85,B 0,C 180,E1 -15566.125,E2 -15566.125} C_VEL
LIN {X 0,Y 312.555,Z 604.812,A -85,B 0,C 180,E1 -15568.71,E2 -15568.71} C_VEL
LIN {X 0,Y 312.773,Z 604.777,A -85,B 0,C 180,E1 -15569.999,E2 -15569.999} C_VEL
LIN {X 0,Y 312.448,Z 603.443,A -85,B 0,C 180,E1 -15572.577,E2 -15572.577} C_VEL
LIN {X 0,Y 312.267,Z 602.202,A -85,B 0,C 180,E1 -15573.87,E2 -15573.87} C_VEL
LIN {X 0,Y 312.147,Z 599.5,A -85,B 0,C 180,E1 -15575.814,E2 -15575.814} C_VEL
LIN {X 0,Y 311.984,Z 595.777,A -85,B 0,C 180,E1 -15577.766,E2 -15577.766} C_VEL
LIN {X 0,Y 311.872,Z 591.086,A -85,B 0,C 180,E1 -15579.729,E2 -15579.729} C_VEL
LIN {X 0,Y 312.06,Z 584.2,A -85,B 0,C 180,E1 -15582.022,E2 -15582.022} C_VEL
LIN {X 0,Y 312.621,Z 575.619,A -85,B 0,C 180,E1 -15584.316,E2 -15584.316} C_VEL
LIN {X 0,Y 313.477,Z 566.674,A -85,B 0,C 180,E1 -15586.273,E2 -15586.273} C_VEL
LIN {X 0,Y 314.775,Z 555.967,A -85,B 0,C 180,E1 -15588.213,E2 -15588.213} C_VEL
LIN {X 0,Y 316.224,Z 543.99,A -85,B 0,C 180,E1 -15589.979,E2 -15589.979} C_VEL
LIN {X 0,Y 317.577,Z 531.727,A -85,B 0,C 180,E1 -15591.461,E2 -15591.461} C_VEL
LIN {X 0,Y 316.759,Z 518.245,A -85,B 0,C 180,E1 -15592.846,E2 -15592.846} C_VEL
LIN {X 0,Y 315.47,Z 503.457,A -85,B 0,C 180,E1 -15594.093,E2 -15594.093} C_VEL
LIN {X 0,Y 314.055,Z 487.681,A -85,B 0,C 180,E1 -15595.121,E2 -15595.121} C_VEL
LIN {X 0,Y 312.778,Z 474.303,A -85,B 0,C 180,E1 -15595.818,E2 -15595.818} C_VEL
LIN {X 0,Y 313.677,Z 464.63,A -85,B 0,C 180,E1 -15599.53,E2 -15599.53} C_VEL
LIN {X 0,Y 314.787,Z 455.281,A -85,B 0,C 180,E1 -15603.159,E2 -15603.159} C_VEL
LIN {X 0,Y 316.054,Z 445.738,A -85,B 0,C 180,E1 -15606.896,E2 -15606.896} C_VEL
LIN {X 0,Y 317.282,Z 438.039,A -85,B 0,C 180,E1 -15609.966,E2 -15609.966} C_VEL
LIN {X 0,Y 317.295,Z 433.995,A -85,B 0,C 180,E1 -15611.641,E2 -15611.641} C_VEL
LIN {X 0,Y 315.517,Z 425.33,A -85,B 0,C 180,E1 -15615.459,E2 -15615.459} C_VEL
LIN {X 0,Y 313.808,Z 416.596,A -85,B 0,C 180,E1 -15619.498,E2 -15619.498} C_VEL
LIN {X 0,Y 312.553,Z 410.178,A -85,B 0,C 180,E1 -15622.619,E2 -15622.619} C_VEL
LIN {X 0,Y 312.51,Z 410.18,A -85,B 0,C 180,E1 -15626.31,E2 -15626.31} C_VEL
LIN {X 0,Y 312.536,Z 410.176,A -85,B 0,C 180,E1 -15630.349,E2 -15630.349} C_VEL
LIN {X 0,Y 312.593,Z 410.169,A -85,B 0,C 180,E1 -15634.064,E2 -15634.064} C_VEL
LIN {X 0,Y 312.577,Z 410.173,A -85,B 0,C 180,E1 -15637.528,E2 -15637.528} C_VEL
LIN {X 0,Y 312.628,Z 410.166,A -85,B 0,C 180,E1 -15641.656,E2 -15641.656} C_VEL
LIN {X 0,Y 312.684,Z 410.158,A -85,B 0,C 180,E1 -15645.686,E2 -15645.686} C_VEL
LIN {X 0,Y 312.693,Z 410.154,A -85,B 0,C 180,E1 -15649.642,E2 -15649.642} C_VEL
LIN {X 0,Y 312.861,Z 410.136,A -85,B 0,C 180,E1 -15652.254,E2 -15652.254} C_VEL
LIN {X 0,Y 312.71,Z 410.158,A -85,B 0,C 180,E1 -15654.843,E2 -15654.843} C_VEL
LIN {X 0,Y 312.943,Z 410.127,A -85,B 0,C 180,E1 -15657.426,E2 -15657.426} C_VEL
LIN {X 0,Y 313.111,Z 410.103,A -85,B 0,C 180,E1 -15660,E2 -15660} C_VEL
LIN {X 0,Y 312.943,Z 410.128,A -85,B 0,C 180,E1 -15662.575,E2 -15662.575} C_VEL
LIN {X 0,Y 312.884,Z 410.131,A -85,B 0,C 180,E1 -15666.647,E2 -15666.647} C_VEL
LIN {X 0,Y 312.778,Z 410.139,A -85,B 0,C 180,E1 -15669.05,E2 -15669.05} C_VEL
LIN {X 0,Y 312.628,Z 410.169,A -85,B 0,C 180,E1 -15672.992,E2 -15672.992} C_VEL
LIN {X 0,Y 312.629,Z 410.164,A -85,B 0,C 180,E1 -15675.651,E2 -15675.651} C_VEL
LIN {X 0,Y 312.622,Z 410.167,A -85,B 0,C 180,E1 -15679.238,E2 -15679.238} C_VEL
LIN {X 0,Y 312.537,Z 410.179,A -85,B 0,C 180,E1 -15682.79,E2 -15682.79} C_VEL
LIN {X 0,Y 312.594,Z 410.169,A -85,B 0,C 180,E1 -15685.937,E2 -15685.937} C_VEL
LIN {X 0,Y 312.537,Z 410.165,A -85,B 0,C 180,E1 -15689.651,E2 -15689.651} C_VEL
LIN {X 0,Y 312.512,Z 410.179,A -85,B 0,C 180,E1 -15693.69,E2 -15693.69} C_VEL
LIN {X 0,Y 312.519,Z 410.172,A -85,B 0,C 180,E1 -15697.387,E2 -15697.387} C_VEL
LIN {X 0,Y 312.484,Z 410.187,A -85,B 0,C 180,E1 -15700.711,E2 -15700.711} C_VEL
LIN {X 0,Y 312.47,Z 410.186,A -85,B 0,C 180,E1 -15704.207,E2 -15704.207} C_VEL
LIN {X 0,Y 312.524,Z 410.179,A -85,B 0,C 180,E1 -15707.911,E2 -15707.911} C_VEL
LIN {X 0,Y 312.554,Z 410.173,A -85,B 0,C 180,E1 -15711.907,E2 -15711.907} C_VEL
LIN {X 0,Y 312.504,Z 410.181,A -85,B 0,C 180,E1 -15715.792,E2 -15715.792} C_VEL
LIN {X 0,Y 312.523,Z 410.178,A -85,B 0,C 180,E1 -15718.856,E2 -15718.856} C_VEL
LIN {X 0,Y 312.572,Z 410.174,A -85,B 0,C 180,E1 -15721.826,E2 -15721.826} C_VEL
LIN {X 0,Y 312.585,Z 410.173,A -85,B 0,C 180,E1 -15724.713,E2 -15724.713} C_VEL
LIN {X 0,Y 312.588,Z 410.174,A -85,B 0,C 180,E1 -15727.531,E2 -15727.531} C_VEL
LIN {X 0,Y 312.605,Z 410.17,A -85,B 0,C 180,E1 -15730.372,E2 -15730.372} C_VEL
LIN {X 0,Y 314.402,Z 414.943,A -85,B 0,C 180,E1 -15730.685,E2 -15730.685} C_VEL
LIN {X 0,Y 318.75,Z 426.343,A -85,B 0,C 180,E1 -15731.522,E2 -15731.522} C_VEL
LIN {X 0,Y 321.782,Z 435.936,A -85,B 0,C 180,E1 -15732.359,E2 -15732.359} C_VEL
LIN {X 0,Y 321.091,Z 448.103,A -85,B 0,C 180,E1 -15733.348,E2 -15733.348} C_VEL
LIN {X 0,Y 320.115,Z 459.666,A -85,B 0,C 180,E1 -15734.563,E2 -15734.563} C_VEL
LIN {X 0,Y 318.922,Z 470.273,A -85,B 0,C 180,E1 -15735.973,E2 -15735.973} C_VEL
LIN {X 0,Y 317.705,Z 479.739,A -85,B 0,C 180,E1 -15737.546,E2 -15737.546} C_VEL
LIN {X 0,Y 316.651,Z 487.495,A -85,B 0,C 180,E1 -15739.127,E2 -15739.127} C_VEL
LIN {X 0,Y 315.454,Z 495.123,A -85,B 0,C 180,E1 -15741.029,E2 -15741.029} C_VEL
LIN {X 0,Y 314.675,Z 501.175,A -85,B 0,C 180,E1 -15742.946,E2 -15742.946} C_VEL
LIN {X 0,Y 313.973,Z 505.988,A -85,B 0,C 180,E1 -15744.865,E2 -15744.865} C_VEL
LIN {X 0,Y 313.38,Z 509.709,A -85,B 0,C 180,E1 -15746.787,E2 -15746.787} C_VEL
LIN {X 0,Y 312.943,Z 512.439,A -85,B 0,C 180,E1 -15748.715,E2 -15748.715} C_VEL
LIN {X 0,Y 312.809,Z 514.613,A -85,B 0,C 180,E1 -15751.289,E2 -15751.289} C_VEL
LIN {X 0,Y 312.705,Z 515.15,A -85,B 0,C 180,E1 -15752.578,E2 -15752.578} C_VEL
LIN {X 0,Y 312.581,Z 515.277,A -85,B 0,C 180,E1 -15753.869,E2 -15753.869} C_VEL
LIN {X 0,Y 313.071,Z 514.336,A -85,B 0,C 180,E1 -15756.446,E2 -15756.446} C_VEL
LIN {X 0,Y 313.492,Z 513.271,A -85,B 0,C 180,E1 -15757.732,E2 -15757.732} C_VEL
LIN {X 0,Y 314.195,Z 509.923,A -85,B 0,C 180,E1 -15760.31,E2 -15760.31} C_VEL
LIN {X 0,Y 315.006,Z 506.248,A -85,B 0,C 180,E1 -15762.238,E2 -15762.238} C_VEL
LIN {X 0,Y 315.847,Z 501.479,A -85,B 0,C 180,E1 -15764.169,E2 -15764.169} C_VEL
LIN {X 0,Y 316.948,Z 495.433,A -85,B 0,C 180,E1 -15766.093,E2 -15766.093} C_VEL
LIN {X 0,Y 318.306,Z 487.798,A -85,B 0,C 180,E1 -15768.007,E2 -15768.007} C_VEL
LIN {X 0,Y 319.89,Z 478.258,A -85,B 0,C 180,E1 -15769.911,E2 -15769.911} C_VEL
LIN {X 0,Y 321.287,Z 468.234,A -85,B 0,C 180,E1 -15771.495,E2 -15771.495} C_VEL
LIN {X 0,Y 322.406,Z 458.321,A -85,B 0,C 180,E1 -15772.765,E2 -15772.765} C_VEL
LIN {X 0,Y 323.403,Z 447.622,A -85,B 0,C 180,E1 -15773.862,E2 -15773.862} C_VEL
LIN {X 0,Y 324.016,Z 440.372,A -85,B 0,C 180,E1 -15774.459,E2 -15774.459} C_VEL
LIN {X 0,Y 322.674,Z 435.247,A -85,B 0,C 180,E1 -15774.971,E2 -15774.971} C_VEL
LIN {X 0,Y 318.373,Z 423.557,A -85,B 0,C 180,E1 -15776.062,E2 -15776.062} C_VEL
LIN {X 0,Y 313.486,Z 412.803,A -85,B 0,C 180,E1 -15776.937,E2 -15776.937} C_VEL
LIN {X 0,Y 312.603,Z 410.172,A -85,B 0,C 180,E1 -15777.134,E2 -15777.134} C_VEL
LIN {X 0,Y 312.523,Z 410.184,A -85,B 0,C 180,E1 -15781.29,E2 -15781.29} C_VEL
LIN {X 0,Y 312.512,Z 410.185,A -85,B 0,C 180,E1 -15784.211,E2 -15784.211} C_VEL
LIN {X 0,Y 312.526,Z 410.169,A -85,B 0,C 180,E1 -15787.386,E2 -15787.386} C_VEL
LIN {X 0,Y 312.496,Z 410.187,A -85,B 0,C 180,E1 -15790.71,E2 -15790.71} C_VEL
LIN {X 0,Y 312.458,Z 410.191,A -85,B 0,C 180,E1 -15794.21,E2 -15794.21} C_VEL
LIN {X 0,Y 312.491,Z 410.186,A -85,B 0,C 180,E1 -15797.919,E2 -15797.919} C_VEL
LIN {X 0,Y 312.504,Z 410.149,A -85,B 0,C 180,E1 -15800.971,E2 -15800.971} C_VEL
LIN {X 0,Y 312.538,Z 410.175,A -85,B 0,C 180,E1 -15804.221,E2 -15804.221} C_VEL
LIN {X 0,Y 312.51,Z 410.173,A -85,B 0,C 180,E1 -15807.334,E2 -15807.334} C_VEL
LIN {X 0,Y 312.549,Z 410.136,A -85,B 0,C 180,E1 -15811.279,E2 -15811.279} C_VEL
LIN {X 0,Y 312.59,Z 410.17,A -85,B 0,C 180,E1 -15814.711,E2 -15814.711} C_VEL
LIN {X 0,Y 312.541,Z 410.18,A -85,B 0,C 180,E1 -15816.176,E2 -15816.176} C_VEL
LIN {X 0,Y 312.475,Z 411.041,A -85,B 0,C 180,E1 -15816.709,E2 -15816.709} C_VEL
LIN {X 0,Y 312.286,Z 413.845,A -85,B 0,C 180,E1 -15817.277,E2 -15817.277} C_VEL
LIN {X 0,Y 311.969,Z 418.793,A -85,B 0,C 180,E1 -15817.802,E2 -15817.802} C_VEL
LIN {X 0,Y 311.673,Z 429.731,A -85,B 0,C 180,E1 -15818.782,E2 -15818.782} C_VEL
LIN {X 0,Y 312.639,Z 436.008,A -85,B 0,C 180,E1 -15819.501,E2 -15819.501} C_VEL
LIN {X 0,Y 313.035,Z 438.555,A -85,B 0,C 180,E1 -15819.806,E2 -15819.806} C_VEL
LIN {X 0,Y 311.793,Z 450.928,A -85,B 0,C 180,E1 -15821.294,E2 -15821.294} C_VEL
LIN {X 0,Y 310.552,Z 462.007,A -85,B 0,C 180,E1 -15822.89,E2 -15822.89} C_VEL
LIN {X 0,Y 309.226,Z 473.305,A -85,B 0,C 180,E1 -15824.848,E2 -15824.848} C_VEL
LIN {X 0,Y 308.294,Z 482.775,A -85,B 0,C 180,E1 -15826.822,E2 -15826.822} C_VEL
LIN {X 0,Y 307.266,Z 491.948,A -85,B 0,C 180,E1 -15829.123,E2 -15829.123} C_VEL
LIN {X 0,Y 306.605,Z 499.469,A -85,B 0,C 180,E1 -15831.431,E2 -15831.431} C_VEL
LIN {X 0,Y 306.132,Z 504.765,A -85,B 0,C 180,E1 -15833.408,E2 -15833.408} C_VEL
LIN {X 0,Y 305.516,Z 510.423,A -85,B 0,C 180,E1 -15836.042,E2 -15836.042} C_VEL
LIN {X 0,Y 305.698,Z 512.647,A -85,B 0,C 180,E1 -15837.364,E2 -15837.364} C_VEL
LIN {X 0,Y 305.797,Z 514.52,A -85,B 0,C 180,E1 -15838.683,E2 -15838.683} C_VEL
LIN {X 0,Y 305.879,Z 517.247,A -85,B 0,C 180,E1 -15841.316,E2 -15841.316} C_VEL
LIN {X 0,Y 306.382,Z 518.618,A -85,B 0,C 180,E1 -15843.946,E2 -15843.946} C_VEL
LIN {X 0,Y 307.19,Z 518.68,A -85,B 0,C 180,E1 -15846.568,E2 -15846.568} C_VEL
LIN {X 0,Y 308.379,Z 517.438,A -85,B 0,C 180,E1 -15849.179,E2 -15849.179} C_VEL
LIN {X 0,Y 310.005,Z 514.878,A -85,B 0,C 180,E1 -15851.773,E2 -15851.773} C_VEL
LIN {X 0,Y 311.939,Z 510.98,A -85,B 0,C 180,E1 -15854.349,E2 -15854.349} C_VEL
LIN {X 0,Y 313.728,Z 507.049,A -85,B 0,C 180,E1 -15856.261,E2 -15856.261} C_VEL
LIN {X 0,Y 316.525,Z 500.478,A -85,B 0,C 180,E1 -15858.781,E2 -15858.781} C_VEL
LIN {X 0,Y 319.433,Z 493.197,A -85,B 0,C 180,E1 -15860.948,E2 -15860.948} C_VEL
LIN {X 0,Y 322.637,Z 484.341,A -85,B 0,C 180,E1 -15863.085,E2 -15863.085} C_VEL
LIN {X 0,Y 325.749,Z 474.958,A -85,B 0,C 180,E1 -15864.947,E2 -15864.947} C_VEL
LIN {X 0,Y 328.978,Z 464.506,A -85,B 0,C 180,E1 -15866.655,E2 -15866.655} C_VEL
LIN {X 0,Y 330.322,Z 459.778,A -85,B 0,C 180,E1 -15867.328,E2 -15867.328} C_VEL
LIN {X 0,Y 329.549,Z 454.606,A -85,B 0,C 180,E1 -15868.553,E2 -15868.553} C_VEL
LIN {X 0,Y 327.703,Z 447.821,A -85,B 0,C 180,E1 -15870.355,E2 -15870.355} C_VEL
LIN {X 0,Y 325.893,Z 442.872,A -85,B 0,C 180,E1 -15871.866,E2 -15871.866} C_VEL
LIN {X 0,Y 324.601,Z 440.46,A -85,B 0,C 180,E1 -15872.771,E2 -15872.771} C_VEL
LIN {X 0,Y 321.658,Z 437.178,A -85,B 0,C 180,E1 -15874.616,E2 -15874.616} C_VEL
LIN {X 0,Y 318.941,Z 434.986,A -85,B 0,C 180,E1 -15876.509,E2 -15876.509} C_VEL
LIN {X 0,Y 316.696,Z 433.734,A -85,B 0,C 180,E1 -15878.416,E2 -15878.416} C_VEL
LIN {X 0,Y 314.666,Z 433.763,A -85,B 0,C 180,E1 -15880.589,E2 -15880.589} C_VEL
LIN {X 0,Y 313.916,Z 433.697,A -85,B 0,C 180,E1 -15882.369,E2 -15882.369} C_VEL
LIN {X 0,Y 313.226,Z 436.782,A -85,B 0,C 180,E1 -15885.201,E2 -15885.201} C_VEL
LIN {X 0,Y 313.964,Z 440.985,A -85,B 0,C 180,E1 -15887.813,E2 -15887.813} C_VEL
LIN {X 0,Y 314.682,Z 443.614,A -85,B 0,C 180,E1 -15889.033,E2 -15889.033} C_VEL
LIN {X 0,Y 315.228,Z 450.587,A -85,B 0,C 180,E1 -15890.781,E2 -15890.781} C_VEL
LIN {X 0,Y 316.012,Z 454.87,A -85,B 0,C 180,E1 -15891.893,E2 -15891.893} C_VEL
LIN {X 0,Y 317.343,Z 463.287,A -85,B 0,C 180,E1 -15893.711,E2 -15893.711} C_VEL
LIN {X 0,Y 318.783,Z 473.054,A -85,B 0,C 180,E1 -15895.54,E2 -15895.54} C_VEL
LIN {X 0,Y 320.128,Z 484.683,A -85,B 0,C 180,E1 -15897.449,E2 -15897.449} C_VEL
LIN {X 0,Y 320.763,Z 496.749,A -85,B 0,C 180,E1 -15899.229,E2 -15899.229} C_VEL
LIN {X 0,Y 320.516,Z 509.493,A -85,B 0,C 180,E1 -15900.983,E2 -15900.983} C_VEL
LIN {X 0,Y 319.209,Z 521.731,A -85,B 0,C 180,E1 -15902.637,E2 -15902.637} C_VEL
LIN {X 0,Y 316.381,Z 537.131,A -85,B 0,C 180,E1 -15904.858,E2 -15904.858} C_VEL
LIN {X 0,Y 314.975,Z 544.024,A -85,B 0,C 180,E1 -15905.969,E2 -15905.969} C_VEL
LIN {X 0,Y 312.004,Z 554.665,A -85,B 0,C 180,E1 -15907.832,E2 -15907.832} C_VEL
LIN {X 0,Y 309.279,Z 565.356,A -85,B 0,C 180,E1 -15910.07,E2 -15910.07} C_VEL
LIN {X 0,Y 307.168,Z 574.443,A -85,B 0,C 180,E1 -15912.351,E2 -15912.351} C_VEL
LIN {X 0,Y 305.537,Z 583.214,A -85,B 0,C 180,E1 -15915.036,E2 -15915.036} C_VEL
LIN {X 0,Y 304.731,Z 589.39,A -85,B 0,C 180,E1 -15917.343,E2 -15917.343} C_VEL
LIN {X 0,Y 304.368,Z 595.107,A -85,B 0,C 180,E1 -15920.026,E2 -15920.026} C_VEL
LIN {X 0,Y 304.452,Z 598.463,A -85,B 0,C 180,E1 -15922.037,E2 -15922.037} C_VEL
LIN {X 0,Y 304.846,Z 601.648,A -85,B 0,C 180,E1 -15924.707,E2 -15924.707} C_VEL
LIN {X 0,Y 305.014,Z 602.679,A -85,B 0,C 180,E1 -15926.035,E2 -15926.035} C_VEL
LIN {X 0,Y 305.54,Z 603.644,A -85,B 0,C 180,E1 -15928.681,E2 -15928.681} C_VEL
LIN {X 0,Y 305.783,Z 603.607,A -85,B 0,C 180,E1 -15929.999,E2 -15929.999} C_VEL
LIN {X 0,Y 305.575,Z 603.22,A -85,B 0,C 180,E1 -15931.316,E2 -15931.316} C_VEL
LIN {X 0,Y 305.392,Z 602.413,A -85,B 0,C 180,E1 -15932.637,E2 -15932.637} C_VEL
LIN {X 0,Y 305.21,Z 601.15,A -85,B 0,C 180,E1 -15933.96,E2 -15933.96} C_VEL
LIN {X 0,Y 305.095,Z 598.451,A -85,B 0,C 180,E1 -15935.948,E2 -15935.948} C_VEL
LIN {X 0,Y 304.909,Z 594.66,A -85,B 0,C 180,E1 -15937.948,E2 -15937.948} C_VEL
LIN {X 0,Y 304.828,Z 589.689,A -85,B 0,C 180,E1 -15939.956,E2 -15939.956} C_VEL
LIN {X 0,Y 305.121,Z 581.239,A -85,B 0,C 180,E1 -15942.638,E2 -15942.638} C_VEL
LIN {X 0,Y 305.815,Z 572.338,A -85,B 0,C 180,E1 -15944.952,E2 -15944.952} C_VEL
LIN {X 0,Y 306.738,Z 562.777,A -85,B 0,C 180,E1 -15946.984,E2 -15946.984} C_VEL
LIN {X 0,Y 308.226,Z 551.484,A -85,B 0,C 180,E1 -15948.959,E2 -15948.959} C_VEL
LIN {X 0,Y 309.674,Z 540.114,A -85,B 0,C 180,E1 -15950.594,E2 -15950.594} C_VEL
LIN {X 0,Y 310.502,Z 531.864,A -85,B 0,C 180,E1 -15951.602,E2 -15951.602} C_VEL
LIN {X 0,Y 309.681,Z 518.355,A -85,B 0,C 180,E1 -15953.045,E2 -15953.045} C_VEL
LIN {X 0,Y 308.483,Z 503.894,A -85,B 0,C 180,E1 -15954.315,E2 -15954.315} C_VEL
LIN {X 0,Y 307.182,Z 488.925,A -85,B 0,C 180,E1 -15955.355,E2 -15955.355} C_VEL
LIN {X 0,Y 305.773,Z 473.409,A -85,B 0,C 180,E1 -15956.201,E2 -15956.201} C_VEL
LIN {X 0,Y 306.78,Z 463.121,A -85,B 0,C 180,E1 -15960.263,E2 -15960.263} C_VEL
LIN {X 0,Y 307.968,Z 453.762,A -85,B 0,C 180,E1 -15963.992,E2 -15963.992} C_VEL
LIN {X 0,Y 309.313,Z 444.251,A -85,B 0,C 180,E1 -15967.839,E2 -15967.839} C_VEL
LIN {X 0,Y 310.288,Z 438.355,A -85,B 0,C 180,E1 -15970.243,E2 -15970.243} C_VEL
LIN {X 0,Y 310.286,Z 435.096,A -85,B 0,C 180,E1 -15971.63,E2 -15971.63} C_VEL
LIN {X 0,Y 308.698,Z 427.346,A -85,B 0,C 180,E1 -15975.109,E2 -15975.109} C_VEL
LIN {X 0,Y 307.033,Z 418.951,A -85,B 0,C 180,E1 -15979.055,E2 -15979.055} C_VEL
LIN {X 0,Y 305.488,Z 411.059,A -85,B 0,C 180,E1 -15983.005,E2 -15983.005} C_VEL
LIN {X 0,Y 305.456,Z 411.059,A -85,B 0,C 180,E1 -15986.482,E2 -15986.482} C_VEL
LIN {X 0,Y 305.487,Z 411.057,A -85,B 0,C 180,E1 -15990.949,E2 -15990.949} C_VEL
LIN {X 0,Y 305.563,Z 411.045,A -85,B 0,C 180,E1 -15994.087,E2 -15994.087} C_VEL
LIN {X 0,Y 305.49,Z 411.055,A -85,B 0,C 180,E1 -15998.402,E2 -15998.402} C_VEL
LIN {X 0,Y 305.58,Z 411.047,A -85,B 0,C 180,E1 -16001.217,E2 -16001.217} C_VEL
LIN {X 0,Y 305.639,Z 411.037,A -85,B 0,C 180,E1 -16005.349,E2 -16005.349} C_VEL
LIN {X 0,Y 305.63,Z 411.035,A -85,B 0,C 180,E1 -16009.4,E2 -16009.4} C_VEL
LIN {X 0,Y 305.802,Z 411.015,A -85,B 0,C 180,E1 -16012.074,E2 -16012.074} C_VEL
LIN {X 0,Y 305.681,Z 411.033,A -85,B 0,C 180,E1 -16014.724,E2 -16014.724} C_VEL
LIN {X 0,Y 305.951,Z 411,A -85,B 0,C 180,E1 -16018.684,E2 -16018.684} C_VEL
LIN {X 0,Y 305.951,Z 410.998,A -85,B 0,C 180,E1 -16021.317,E2 -16021.317} C_VEL
LIN {X 0,Y 305.682,Z 411.03,A -85,B 0,C 180,E1 -16025.277,E2 -16025.277} C_VEL
LIN {X 0,Y 305.803,Z 411.007,A -85,B 0,C 180,E1 -16027.926,E2 -16027.926} C_VEL
LIN {X 0,Y 305.597,Z 411.038,A -85,B 0,C 180,E1 -16031.946,E2 -16031.946} C_VEL
LIN {X 0,Y 305.628,Z 411.039,A -85,B 0,C 180,E1 -16035.036,E2 -16035.036} C_VEL
LIN {X 0,Y 305.568,Z 411.045,A -85,B 0,C 180,E1 -16039.446,E2 -16039.446} C_VEL
LIN {X 0,Y 305.482,Z 411.057,A -85,B 0,C 180,E1 -16043.042,E2 -16043.042} C_VEL
LIN {X 0,Y 305.539,Z 411.049,A -85,B 0,C 180,E1 -16046.228,E2 -16046.228} C_VEL
LIN {X 0,Y 305.487,Z 411.044,A -85,B 0,C 180,E1 -16049.051,E2 -16049.051} C_VEL
LIN {X 0,Y 305.458,Z 411.058,A -85,B 0,C 180,E1 -16053.518,E2 -16053.518} C_VEL
LIN {X 0,Y 305.468,Z 411.054,A -85,B 0,C 180,E1 -16056.741,E2 -16056.741} C_VEL
LIN {X 0,Y 305.449,Z 411.061,A -85,B 0,C 180,E1 -16060.601,E2 -16060.601} C_VEL
LIN {X 0,Y 305.42,Z 411.061,A -85,B 0,C 180,E1 -16064.496,E2 -16064.496} C_VEL
LIN {X 0,Y 305.472,Z 411.059,A -85,B 0,C 180,E1 -16068.151,E2 -16068.151} C_VEL
LIN {X 0,Y 305.515,Z 411.049,A -85,B 0,C 180,E1 -16071.606,E2 -16071.606} C_VEL
LIN {X 0,Y 305.461,Z 411.06,A -85,B 0,C 180,E1 -16074.889,E2 -16074.889} C_VEL
LIN {X 0,Y 305.451,Z 411.061,A -85,B 0,C 180,E1 -16078.356,E2 -16078.356} C_VEL
LIN {X 0,Y 305.518,Z 411.052,A -85,B 0,C 180,E1 -16081.116,E2 -16081.116} C_VEL
LIN {X 0,Y 305.57,Z 411.049,A -85,B 0,C 180,E1 -16084.09,E2 -16084.09} C_VEL
LIN {X 0,Y 305.501,Z 411.059,A -85,B 0,C 180,E1 -16088.405,E2 -16088.405} C_VEL
LIN {X 0,Y 305.538,Z 411.053,A -85,B 0,C 180,E1 -16089.875,E2 -16089.875} C_VEL
LIN {X 0,Y 306.55,Z 413.933,A -85,B 0,C 180,E1 -16090.048,E2 -16090.048} C_VEL
LIN {X 0,Y 311.024,Z 425.036,A -85,B 0,C 180,E1 -16090.869,E2 -16090.869} C_VEL
LIN {X 0,Y 314.758,Z 436.33,A -85,B 0,C 180,E1 -16091.863,E2 -16091.863} C_VEL
LIN {X 0,Y 315.108,Z 439.482,A -85,B 0,C 180,E1 -16092.134,E2 -16092.134} C_VEL
LIN {X 0,Y 314.303,Z 450.745,A -85,B 0,C 180,E1 -16093.103,E2 -16093.103} C_VEL
LIN {X 0,Y 313.252,Z 462.277,A -85,B 0,C 180,E1 -16094.383,E2 -16094.383} C_VEL
LIN {X 0,Y 311.968,Z 472.698,A -85,B 0,C 180,E1 -16095.846,E2 -16095.846} C_VEL
LIN {X 0,Y 310.606,Z 482.649,A -85,B 0,C 180,E1 -16097.589,E2 -16097.589} C_VEL
LIN {X 0,Y 309.335,Z 491.373,A -85,B 0,C 180,E1 -16099.529,E2 -16099.529} C_VEL
LIN {X 0,Y 308.231,Z 498.407,A -85,B 0,C 180,E1 -16101.479,E2 -16101.479} C_VEL
LIN {X 0,Y 307.494,Z 504.015,A -85,B 0,C 180,E1 -16103.439,E2 -16103.439} C_VEL
LIN {X 0,Y 306.777,Z 508.44,A -85,B 0,C 180,E1 -16105.402,E2 -16105.402} C_VEL
LIN {X 0,Y 306.16,Z 511.808,A -85,B 0,C 180,E1 -16107.37,E2 -16107.37} C_VEL
LIN {X 0,Y 305.92,Z 513.486,A -85,B 0,C 180,E1 -16108.685,E2 -16108.685} C_VEL
LIN {X 0,Y 305.788,Z 515.64,A -85,B 0,C 180,E1 -16111.318,E2 -16111.318} C_VEL
LIN {X 0,Y 305.681,Z 516.162,A -85,B 0,C 180,E1 -16112.637,E2 -16112.637} C_VEL
LIN {X 0,Y 305.561,Z 516.278,A -85,B 0,C 180,E1 -16113.958,E2 -16113.958} C_VEL
LIN {X 0,Y 306.083,Z 515.316,A -85,B 0,C 180,E1 -16116.594,E2 -16116.594} C_VEL
LIN {X 0,Y 306.524,Z 514.232,A -85,B 0,C 180,E1 -16117.909,E2 -16117.909} C_VEL
LIN {X 0,Y 307.183,Z 511.202,A -85,B 0,C 180,E1 -16120.327,E2 -16120.327} C_VEL
LIN {X 0,Y 308.131,Z 507.167,A -85,B 0,C 180,E1 -16122.515,E2 -16122.515} C_VEL
LIN {X 0,Y 309.023,Z 502.375,A -85,B 0,C 180,E1 -16124.489,E2 -16124.489} C_VEL
LIN {X 0,Y 310.173,Z 496.295,A -85,B 0,C 180,E1 -16126.454,E2 -16126.454} C_VEL
LIN {X 0,Y 311.602,Z 488.624,A -85,B 0,C 180,E1 -16128.408,E2 -16128.408} C_VEL
LIN {X 0,Y 313.268,Z 479.038,A -85,B 0,C 180,E1 -16130.35,E2 -16130.35} C_VEL
LIN {X 0,Y 314.716,Z 468.955,A -85,B 0,C 180,E1 -16131.967,E2 -16131.967} C_VEL
LIN {X 0,Y 315.901,Z 458.977,A -85,B 0,C 180,E1 -16133.261,E2 -16133.261} C_VEL
LIN {X 0,Y 316.948,Z 448.194,A -85,B 0,C 180,E1 -16134.379,E2 -16134.379} C_VEL
LIN {X 0,Y 317.473,Z 442.341,A -85,B 0,C 180,E1 -16134.874,E2 -16134.874} C_VEL
LIN {X 0,Y 316.38,Z 437.785,A -85,B 0,C 180,E1 -16135.345,E2 -16135.345} C_VEL
LIN {X 0,Y 312.138,Z 426.178,A -85,B 0,C 180,E1 -16136.491,E2 -16136.491} C_VEL
LIN {X 0,Y 306.827,Z 414.284,A -85,B 0,C 180,E1 -16137.506,E2 -16137.506} C_VEL
LIN {X 0,Y 305.682,Z 411.796,A -85,B 0,C 180,E1 -16137.693,E2 -16137.693} C_VEL
LIN {X 0,Y 305.534,Z 411.052,A -85,B 0,C 180,E1 -16137.764,E2 -16137.764} C_VEL
LIN {X 0,Y 305.45,Z 411.066,A -85,B 0,C 180,E1 -16141.953,E2 -16141.953} C_VEL
LIN {X 0,Y 305.468,Z 411.062,A -85,B 0,C 180,E1 -16145.114,E2 -16145.114} C_VEL
LIN {X 0,Y 305.446,Z 411.046,A -85,B 0,C 180,E1 -16148.527,E2 -16148.527} C_VEL
LIN {X 0,Y 305.461,Z 411.057,A -85,B 0,C 180,E1 -16152.586,E2 -16152.586} C_VEL
LIN {X 0,Y 305.441,Z 411.059,A -85,B 0,C 180,E1 -16156.347,E2 -16156.347} C_VEL
LIN {X 0,Y 305.464,Z 411.035,A -85,B 0,C 180,E1 -16159.893,E2 -16159.893} C_VEL
LIN {X 0,Y 305.486,Z 411.047,A -85,B 0,C 180,E1 -16163.632,E2 -16163.632} C_VEL
LIN {X 0,Y 305.471,Z 411.056,A -85,B 0,C 180,E1 -16166.483,E2 -16166.483} C_VEL
LIN {X 0,Y 305.463,Z 411.017,A -85,B 0,C 180,E1 -16169.59,E2 -16169.59} C_VEL
LIN {X 0,Y 305.524,Z 411.029,A -85,B 0,C 180,E1 -16172.608,E2 -16172.608} C_VEL
LIN {X 0,Y 305.517,Z 411.054,A -85,B 0,C 180,E1 -16176.186,E2 -16176.186} C_VEL
LIN {X 0,Y 305.51,Z 411.054,A -85,B 0,C 180,E1 -16176.818,E2 -16176.818} C_VEL
LIN {X 0,Y 309.958,Z 426.436,A -85,B 0,C 180,E1 -16178.38,E2 -16178.38} C_VEL
LIN {X 0,Y 312.639,Z 436.008,A -85,B 0,C 180,E1 -16179.501,E2 -16179.501} C_VEL
LIN {X 0,Y 312.941,Z 439.308,A -85,B 0,C 180,E1 -16179.886,E2 -16179.886} C_VEL
LIN {X 0,Y 312.315,Z 442.59,A -85,B 0,C 180,E1 -16180.247,E2 -16180.247} C_VEL
LIN {X 0,Y 311.061,Z 445.862,A -85,B 0,C 180,E1 -16180.585,E2 -16180.585} C_VEL
LIN {X 0,Y 305.107,Z 456.968,A -85,B 0,C 180,E1 -16181.837,E2 -16181.837} C_VEL
LIN {X 0,Y 303.71,Z 461.641,A -85,B 0,C 180,E1 -16182.508,E2 -16182.508} C_VEL
LIN {X 0,Y 302.336,Z 473.148,A -85,B 0,C 180,E1 -16184.494,E2 -16184.494} C_VEL
LIN {X 0,Y 301.351,Z 482.811,A -85,B 0,C 180,E1 -16186.513,E2 -16186.513} C_VEL
LIN {X 0,Y 300.288,Z 492.17,A -85,B 0,C 180,E1 -16188.867,E2 -16188.867} C_VEL
LIN {X 0,Y 299.575,Z 499.853,A -85,B 0,C 180,E1 -16191.228,E2 -16191.228} C_VEL
LIN {X 0,Y 299.11,Z 505.296,A -85,B 0,C 180,E1 -16193.253,E2 -16193.253} C_VEL
LIN {X 0,Y 298.473,Z 511.11,A -85,B 0,C 180,E1 -16195.949,E2 -16195.949} C_VEL
LIN {X 0,Y 298.775,Z 515.356,A -85,B 0,C 180,E1 -16198.652,E2 -16198.652} C_VEL
LIN {X 0,Y 298.859,Z 518.273,A -85,B 0,C 180,E1 -16201.347,E2 -16201.347} C_VEL
LIN {X 0,Y 299.421,Z 519.812,A -85,B 0,C 180,E1 -16204.038,E2 -16204.038} C_VEL
LIN {X 0,Y 300.264,Z 520.034,A -85,B 0,C 180,E1 -16206.72,E2 -16206.72} C_VEL
LIN {X 0,Y 301.544,Z 518.955,A -85,B 0,C 180,E1 -16209.389,E2 -16209.389} C_VEL
LIN {X 0,Y 303.272,Z 516.569,A -85,B 0,C 180,E1 -16212.038,E2 -16212.038} C_VEL
LIN {X 0,Y 305.326,Z 512.866,A -85,B 0,C 180,E1 -16214.667,E2 -16214.667} C_VEL
LIN {X 0,Y 307.939,Z 507.72,A -85,B 0,C 180,E1 -16217.259,E2 -16217.259} C_VEL
LIN {X 0,Y 311.001,Z 500.963,A -85,B 0,C 180,E1 -16219.814,E2 -16219.814} C_VEL
LIN {X 0,Y 314.643,Z 492.399,A -85,B 0,C 180,E1 -16222.316,E2 -16222.316} C_VEL
LIN {X 0,Y 318.239,Z 483.084,A -85,B 0,C 180,E1 -16224.489,E2 -16224.489} C_VEL
LIN {X 0,Y 321.847,Z 472.722,A -85,B 0,C 180,E1 -16226.452,E2 -16226.452} C_VEL
LIN {X 0,Y 325.06,Z 462.587,A -85,B 0,C 180,E1 -16228.047,E2 -16228.047} C_VEL
LIN {X 0,Y 323.836,Z 455.518,A -85,B 0,C 180,E1 -16229.944,E2 -16229.944} C_VEL
LIN {X 0,Y 321.803,Z 448.473,A -85,B 0,C 180,E1 -16232.14,E2 -16232.14} C_VEL
LIN {X 0,Y 320.407,Z 445.833,A -85,B 0,C 180,E1 -16233.255,E2 -16233.255} C_VEL
LIN {X 0,Y 317.821,Z 442.962,A -85,B 0,C 180,E1 -16235.095,E2 -16235.095} C_VEL
LIN {X 0,Y 315.425,Z 441.112,A -85,B 0,C 180,E1 -16236.984,E2 -16236.984} C_VEL
LIN {X 0,Y 313.942,Z 440.281,A -85,B 0,C 180,E1 -16238.415,E2 -16238.415} C_VEL
LIN {X 0,Y 311.958,Z 440.34,A -85,B 0,C 180,E1 -16240.793,E2 -16240.793} C_VEL
LIN {X 0,Y 311.525,Z 440.342,A -85,B 0,C 180,E1 -16241.884,E2 -16241.884} C_VEL
LIN {X 0,Y 311.234,Z 440.713,A -85,B 0,C 180,E1 -16242.643,E2 -16242.643} C_VEL
LIN {X 0,Y 310.743,Z 444.012,A -85,B 0,C 180,E1 -16245.482,E2 -16245.482} C_VEL
LIN {X 0,Y 311.204,Z 447.029,A -85,B 0,C 180,E1 -16247.35,E2 -16247.35} C_VEL
LIN {X 0,Y 311.707,Z 449.65,A -85,B 0,C 180,E1 -16248.546,E2 -16248.546} C_VEL
LIN {X 0,Y 311.837,Z 455.338,A -85,B 0,C 180,E1 -16250.02,E2 -16250.02} C_VEL
LIN {X 0,Y 312.289,Z 458.573,A -85,B 0,C 180,E1 -16250.939,E2 -16250.939} C_VEL
LIN {X 0,Y 313.267,Z 467.637,A -85,B 0,C 180,E1 -16253.011,E2 -16253.011} C_VEL
LIN {X 0,Y 314.338,Z 477.901,A -85,B 0,C 180,E1 -16255.034,E2 -16255.034} C_VEL
LIN {X 0,Y 315.134,Z 489.638,A -85,B 0,C 180,E1 -16257.034,E2 -16257.034} C_VEL
LIN {X 0,Y 315.271,Z 501.15,A -85,B 0,C 180,E1 -16258.827,E2 -16258.827} C_VEL
LIN {X 0,Y 314.559,Z 513.371,A -85,B 0,C 180,E1 -16260.616,E2 -16260.616} C_VEL
LIN {X 0,Y 312.694,Z 525.678,A -85,B 0,C 180,E1 -16262.382,E2 -16262.382} C_VEL
LIN {X 0,Y 309.862,Z 539.098,A -85,B 0,C 180,E1 -16264.472,E2 -16264.472} C_VEL
LIN {X 0,Y 308.012,Z 546.536,A -85,B 0,C 180,E1 -16265.749,E2 -16265.749} C_VEL
LIN {X 0,Y 305.007,Z 556.564,A -85,B 0,C 180,E1 -16267.653,E2 -16267.653} C_VEL
LIN {X 0,Y 301.865,Z 568.032,A -85,B 0,C 180,E1 -16270.269,E2 -16270.269} C_VEL
LIN {X 0,Y 299.615,Z 577.525,A -85,B 0,C 180,E1 -16272.948,E2 -16272.948} C_VEL
LIN {X 0,Y 298.128,Z 585.362,A -85,B 0,C 180,E1 -16275.668,E2 -16275.668} C_VEL
LIN {X 0,Y 297.451,Z 591.674,A -85,B 0,C 180,E1 -16278.413,E2 -16278.413} C_VEL
LIN {X 0,Y 297.318,Z 596.519,A -85,B 0,C 180,E1 -16281.16,E2 -16281.16} C_VEL
LIN {X 0,Y 297.547,Z 599.234,A -85,B 0,C 180,E1 -16283.216,E2 -16283.216} C_VEL
LIN {X 0,Y 297.785,Z 600.585,A -85,B 0,C 180,E1 -16284.582,E2 -16284.582} C_VEL
LIN {X 0,Y 298.156,Z 602.172,A -85,B 0,C 180,E1 -16287.296,E2 -16287.296} C_VEL
LIN {X 0,Y 298.523,Z 602.509,A -85,B 0,C 180,E1 -16288.65,E2 -16288.65} C_VEL
LIN {X 0,Y 298.755,Z 602.579,A -85,B 0,C 180,E1 -16289.999,E2 -16289.999} C_VEL
LIN {X 0,Y 298.541,Z 602.192,A -85,B 0,C 180,E1 -16291.347,E2 -16291.347} C_VEL
LIN {X 0,Y 298.335,Z 601.378,A -85,B 0,C 180,E1 -16292.699,E2 -16292.699} C_VEL
LIN {X 0,Y 298.156,Z 600.098,A -85,B 0,C 180,E1 -16294.054,E2 -16294.054} C_VEL
LIN {X 0,Y 298.019,Z 597.381,A -85,B 0,C 180,E1 -16296.09,E2 -16296.09} C_VEL
LIN {X 0,Y 297.82,Z 593.569,A -85,B 0,C 180,E1 -16298.138,E2 -16298.138} C_VEL
LIN {X 0,Y 297.769,Z 588.583,A -85,B 0,C 180,E1 -16300.194,E2 -16300.194} C_VEL
LIN {X 0,Y 297.933,Z 582.291,A -85,B 0,C 180,E1 -16302.256,E2 -16302.256} C_VEL
LIN {X 0,Y 298.496,Z 574.48,A -85,B 0,C 180,E1 -16304.311,E2 -16304.311} C_VEL
LIN {X 0,Y 299.564,Z 563.928,A -85,B 0,C 180,E1 -16306.7,E2 -16306.7} C_VEL
LIN {X 0,Y 300.653,Z 555.014,A -85,B 0,C 180,E1 -16308.394,E2 -16308.394} C_VEL
LIN {X 0,Y 302.116,Z 543.382,A -85,B 0,C 180,E1 -16310.243,E2 -16310.243} C_VEL
LIN {X 0,Y 303.436,Z 531.845,A -85,B 0,C 180,E1 -16311.75,E2 -16311.75} C_VEL
LIN {X 0,Y 302.737,Z 520.054,A -85,B 0,C 180,E1 -16313.079,E2 -16313.079} C_VEL
LIN {X 0,Y 301.565,Z 505.406,A -85,B 0,C 180,E1 -16314.447,E2 -16314.447} C_VEL
LIN {X 0,Y 300.293,Z 490.421,A -85,B 0,C 180,E1 -16315.561,E2 -16315.561} C_VEL
LIN {X 0,Y 298.895,Z 474.894,A -85,B 0,C 180,E1 -16316.439,E2 -16316.439} C_VEL
LIN {X 0,Y 298.767,Z 472.51,A -85,B 0,C 180,E1 -16316.592,E2 -16316.592} C_VEL
LIN {X 0,Y 299.922,Z 461.596,A -85,B 0,C 180,E1 -16321.03,E2 -16321.03} C_VEL
LIN {X 0,Y 301.317,Z 451.227,A -85,B 0,C 180,E1 -16325.279,E2 -16325.279} C_VEL
LIN {X 0,Y 302.938,Z 441.228,A -85,B 0,C 180,E1 -16329.448,E2 -16329.448} C_VEL
LIN {X 0,Y 303.346,Z 437.03,A -85,B 0,C 180,E1 -16331.237,E2 -16331.237} C_VEL
LIN {X 0,Y 302.092,Z 430.368,A -85,B 0,C 180,E1 -16334.259,E2 -16334.259} C_VEL
LIN {X 0,Y 300.3,Z 421.468,A -85,B 0,C 180,E1 -16338.493,E2 -16338.493} C_VEL
LIN {X 0,Y 298.819,Z 413.853,A -85,B 0,C 180,E1 -16342.302,E2 -16342.302} C_VEL
LIN {X 0,Y 298.47,Z 411.933,A -85,B 0,C 180,E1 -16343.366,E2 -16343.366} C_VEL
LIN {X 0,Y 298.386,Z 411.942,A -85,B 0,C 180,E1 -16347.199,E2 -16347.199} C_VEL
LIN {X 0,Y 298.46,Z 411.93,A -85,B 0,C 180,E1 -16351.904,E2 -16351.904} C_VEL
LIN {X 0,Y 298.476,Z 411.93,A -85,B 0,C 180,E1 -16354.923,E2 -16354.923} C_VEL
LIN {X 0,Y 298.439,Z 411.933,A -85,B 0,C 180,E1 -16359.315,E2 -16359.315} C_VEL
LIN {X 0,Y 298.528,Z 411.922,A -85,B 0,C 180,E1 -16362.179,E2 -16362.179} C_VEL
LIN {X 0,Y 298.583,Z 411.916,A -85,B 0,C 180,E1 -16364.995,E2 -16364.995} C_VEL
LIN {X 0,Y 298.585,Z 411.914,A -85,B 0,C 180,E1 -16369.147,E2 -16369.147} C_VEL
LIN {X 0,Y 298.748,Z 411.894,A -85,B 0,C 180,E1 -16371.886,E2 -16371.886} C_VEL
LIN {X 0,Y 298.652,Z 411.908,A -85,B 0,C 180,E1 -16374.599,E2 -16374.599} C_VEL
LIN {X 0,Y 298.918,Z 411.876,A -85,B 0,C 180,E1 -16378.653,E2 -16378.653} C_VEL
LIN {X 0,Y 298.918,Z 411.873,A -85,B 0,C 180,E1 -16381.348,E2 -16381.348} C_VEL
LIN {X 0,Y 298.653,Z 411.905,A -85,B 0,C 180,E1 -16385.402,E2 -16385.402} C_VEL
LIN {X 0,Y 298.748,Z 411.885,A -85,B 0,C 180,E1 -16388.115,E2 -16388.115} C_VEL
LIN {X 0,Y 298.547,Z 411.917,A -85,B 0,C 180,E1 -16392.232,E2 -16392.232} C_VEL
LIN {X 0,Y 298.597,Z 411.914,A -85,B 0,C 180,E1 -16395.21,E2 -16395.21} C_VEL
LIN {X 0,Y 298.531,Z 411.923,A -85,B 0,C 180,E1 -16399.244,E2 -16399.244} C_VEL
LIN {X 0,Y 298.449,Z 411.931,A -85,B 0,C 180,E1 -16403.599,E2 -16403.599} C_VEL
LIN {X 0,Y 298.482,Z 411.929,A -85,B 0,C 180,E1 -16406.576,E2 -16406.576} C_VEL
LIN {X 0,Y 298.413,Z 411.922,A -85,B 0,C 180,E1 -16409.642,E2 -16409.642} C_VEL
LIN {X 0,Y 298.388,Z 411.942,A -85,B 0,C 180,E1 -16412.802,E2 -16412.802} C_VEL
LIN {X 0,Y 298.44,Z 411.928,A -85,B 0,C 180,E1 -16416.809,E2 -16416.809} C_VEL
LIN {X 0,Y 298.382,Z 411.941,A -85,B 0,C 180,E1 -16421.089,E2 -16421.089} C_VEL
LIN {X 0,Y 298.384,Z 411.934,A -85,B 0,C 180,E1 -16425.043,E2 -16425.043} C_VEL
LIN {X 0,Y 298.414,Z 411.937,A -85,B 0,C 180,E1 -16428.907,E2 -16428.907} C_VEL
LIN {X 0,Y 298.468,Z 411.93,A -85,B 0,C 180,E1 -16433.188,E2 -16433.188} C_VEL
LIN {X 0,Y 298.394,Z 411.939,A -85,B 0,C 180,E1 -16437.202,E2 -16437.202} C_VEL
LIN {X 0,Y 298.43,Z 411.938,A -85,B 0,C 180,E1 -16440.617,E2 -16440.617} C_VEL
LIN {X 0,Y 298.482,Z 411.929,A -85,B 0,C 180,E1 -16443.476,E2 -16443.476} C_VEL
LIN {X 0,Y 298.436,Z 411.939,A -85,B 0,C 180,E1 -16446.699,E2 -16446.699} C_VEL
LIN {X 0,Y 298.451,Z 411.935,A -85,B 0,C 180,E1 -16449.317,E2 -16449.317} C_VEL
LIN {X 0,Y 300.103,Z 416.342,A -85,B 0,C 180,E1 -16449.609,E2 -16449.609} C_VEL
LIN {X 0,Y 304.49,Z 426.926,A -85,B 0,C 180,E1 -16450.449,E2 -16450.449} C_VEL
LIN {X 0,Y 308.378,Z 438.912,A -85,B 0,C 180,E1 -16451.56,E2 -16451.56} C_VEL
LIN {X 0,Y 308.014,Z 446.928,A -85,B 0,C 180,E1 -16452.228,E2 -16452.228} C_VEL
LIN {X 0,Y 307.067,Z 458.228,A -85,B 0,C 180,E1 -16453.377,E2 -16453.377} C_VEL
LIN {X 0,Y 305.804,Z 469.533,A -85,B 0,C 180,E1 -16454.852,E2 -16454.852} C_VEL
LIN {X 0,Y 304.533,Z 479.066,A -85,B 0,C 180,E1 -16456.399,E2 -16456.399} C_VEL
LIN {X 0,Y 303.285,Z 486.968,A -85,B 0,C 180,E1 -16457.964,E2 -16457.964} C_VEL
LIN {X 0,Y 302.053,Z 495.039,A -85,B 0,C 180,E1 -16459.952,E2 -16459.952} C_VEL
LIN {X 0,Y 300.912,Z 501.543,A -85,B 0,C 180,E1 -16461.946,E2 -16461.946} C_VEL
LIN {X 0,Y 300.291,Z 506.685,A -85,B 0,C 180,E1 -16463.956,E2 -16463.956} C_VEL
LIN {X 0,Y 299.519,Z 510.732,A -85,B 0,C 180,E1 -16465.965,E2 -16465.965} C_VEL
LIN {X 0,Y 299.144,Z 512.871,A -85,B 0,C 180,E1 -16467.308,E2 -16467.308} C_VEL
LIN {X 0,Y 298.791,Z 515.788,A -85,B 0,C 180,E1 -16470.001,E2 -16470.001} C_VEL
LIN {X 0,Y 298.767,Z 516.667,A -85,B 0,C 180,E1 -16471.349,E2 -16471.349} C_VEL
LIN {X 0,Y 298.657,Z 517.172,A -85,B 0,C 180,E1 -16472.699,E2 -16472.699} C_VEL
LIN {X 0,Y 298.541,Z 517.278,A -85,B 0,C 180,E1 -16474.051,E2 -16474.051} C_VEL
LIN {X 0,Y 299.099,Z 516.297,A -85,B 0,C 180,E1 -16476.748,E2 -16476.748} C_VEL
LIN {X 0,Y 299.559,Z 515.193,A -85,B 0,C 180,E1 -16478.094,E2 -16478.094} C_VEL
LIN {X 0,Y 300.27,Z 512.145,A -85,B 0,C 180,E1 -16480.565,E2 -16480.565} C_VEL
LIN {X 0,Y 301.265,Z 508.086,A -85,B 0,C 180,E1 -16482.805,E2 -16482.805} C_VEL
LIN {X 0,Y 302.212,Z 503.271,A -85,B 0,C 180,E1 -16484.823,E2 -16484.823} C_VEL
LIN {X 0,Y 303.402,Z 497.155,A -85,B 0,C 180,E1 -16486.832,E2 -16486.832} C_VEL
LIN {X 0,Y 304.914,Z 489.45,A -85,B 0,C 180,E1 -16488.827,E2 -16488.827} C_VEL
LIN {X 0,Y 306.668,Z 479.813,A -85,B 0,C 180,E1 -16490.808,E2 -16490.808} C_VEL
LIN {X 0,Y 308.191,Z 469.674,A -85,B 0,C 180,E1 -16492.457,E2 -16492.457} C_VEL
LIN {X 0,Y 309.418,Z 459.636,A -85,B 0,C 180,E1 -16493.778,E2 -16493.778} C_VEL
LIN {X 0,Y 310.566,Z 448.39,A -85,B 0,C 180,E1 -16494.95,E2 -16494.95} C_VEL
LIN {X 0,Y 310.95,Z 444.303,A -85,B 0,C 180,E1 -16495.301,E2 -16495.301} C_VEL
LIN {X 0,Y 310.641,Z 442.116,A -85,B 0,C 180,E1 -16495.52,E2 -16495.52} C_VEL
LIN {X 0,Y 306.684,Z 430.675,A -85,B 0,C 180,E1 -16496.745,E2 -16496.745} C_VEL
LIN {X 0,Y 301.796,Z 419.415,A -85,B 0,C 180,E1 -16497.809,E2 -16497.809} C_VEL
LIN {X 0,Y 298.686,Z 412.832,A -85,B 0,C 180,E1 -16498.347,E2 -16498.347} C_VEL
LIN {X 0,Y 298.512,Z 411.927,A -85,B 0,C 180,E1 -16498.412,E2 -16498.412} C_VEL
LIN {X 0,Y 298.402,Z 411.942,A -85,B 0,C 180,E1 -16502.801,E2 -16502.801} C_VEL
LIN {X 0,Y 298.45,Z 411.929,A -85,B 0,C 180,E1 -16506.808,E2 -16506.808} C_VEL
LIN {X 0,Y 298.393,Z 411.941,A -85,B 0,C 180,E1 -16511.088,E2 -16511.088} C_VEL
LIN {X 0,Y 298.404,Z 411.938,A -85,B 0,C 180,E1 -16513.104,E2 -16513.104} C_VEL
LIN {X 0,Y 298.409,Z 411.939,A -85,B 0,C 180,E1 -16516.921,E2 -16516.921} C_VEL
LIN {X 0,Y 298.404,Z 411.904,A -85,B 0,C 180,E1 -16521.008,E2 -16521.008} C_VEL
LIN {X 0,Y 298.424,Z 411.929,A -85,B 0,C 180,E1 -16523.93,E2 -16523.93} C_VEL
LIN {X 0,Y 298.399,Z 411.92,A -85,B 0,C 180,E1 -16527.984,E2 -16527.984} C_VEL
LIN {X 0,Y 298.464,Z 411.896,A -85,B 0,C 180,E1 -16531.904,E2 -16531.904} C_VEL
LIN {X 0,Y 298.489,Z 411.927,A -85,B 0,C 180,E1 -16534.924,E2 -16534.924} C_VEL
LIN {X 0,Y 298.468,Z 411.932,A -85,B 0,C 180,E1 -16536.492,E2 -16536.492} C_VEL
LIN {X 0,Y 302.632,Z 426.404,A -85,B 0,C 180,E1 -16537.982,E2 -16537.982} C_VEL
LIN {X 0,Y 306.113,Z 439.295,A -85,B 0,C 180,E1 -16539.534,E2 -16539.534} C_VEL
LIN {X 0,Y 304.774,Z 452.523,A -85,B 0,C 180,E1 -16541.165,E2 -16541.165} C_VEL
LIN {X 0,Y 303.71,Z 461.641,A -85,B 0,C 180,E1 -16542.508,E2 -16542.508} C_VEL
LIN {X 0,Y 302.575,Z 466.127,A -85,B 0,C 180,E1 -16543.201,E2 -16543.201} C_VEL
LIN {X 0,Y 298.997,Z 473.187,A -85,B 0,C 180,E1 -16544.337,E2 -16544.337} C_VEL
LIN {X 0,Y 295.418,Z 479.853,A -85,B 0,C 180,E1 -16545.574,E2 -16545.574} C_VEL
LIN {X 0,Y 294.302,Z 483.725,A -85,B 0,C 180,E1 -16546.415,E2 -16546.415} C_VEL
LIN {X 0,Y 293.315,Z 492.339,A -85,B 0,C 180,E1 -16548.599,E2 -16548.599} C_VEL
LIN {X 0,Y 292.545,Z 500.203,A -85,B 0,C 180,E1 -16551.016,E2 -16551.016} C_VEL
LIN {X 0,Y 292.091,Z 505.802,A -85,B 0,C 180,E1 -16553.09,E2 -16553.09} C_VEL
LIN {X 0,Y 291.432,Z 511.766,A -85,B 0,C 180,E1 -16555.851,E2 -16555.851} C_VEL
LIN {X 0,Y 291.752,Z 516.172,A -85,B 0,C 180,E1 -16558.619,E2 -16558.619} C_VEL
LIN {X 0,Y 291.838,Z 519.245,A -85,B 0,C 180,E1 -16561.38,E2 -16561.38} C_VEL
LIN {X 0,Y 292.429,Z 520.969,A -85,B 0,C 180,E1 -16564.134,E2 -16564.134} C_VEL
LIN {X 0,Y 293.34,Z 521.386,A -85,B 0,C 180,E1 -16566.88,E2 -16566.88} C_VEL
LIN {X 0,Y 294.706,Z 520.495,A -85,B 0,C 180,E1 -16569.609,E2 -16569.609} C_VEL
LIN {X 0,Y 296.557,Z 518.29,A -85,B 0,C 180,E1 -16572.315,E2 -16572.315} C_VEL
LIN {X 0,Y 298.723,Z 514.793,A -85,B 0,C 180,E1 -16574.998,E2 -16574.998} C_VEL
LIN {X 0,Y 301.506,Z 509.866,A -85,B 0,C 180,E1 -16577.639,E2 -16577.639} C_VEL
LIN {X 0,Y 304.751,Z 503.453,A -85,B 0,C 180,E1 -16580.238,E2 -16580.238} C_VEL
LIN {X 0,Y 308.581,Z 495.212,A -85,B 0,C 180,E1 -16582.779,E2 -16582.779} C_VEL
LIN {X 0,Y 312.317,Z 486.416,A -85,B 0,C 180,E1 -16584.956,E2 -16584.956} C_VEL
LIN {X 0,Y 315.863,Z 477.353,A -85,B 0,C 180,E1 -16586.796,E2 -16586.796} C_VEL
LIN {X 0,Y 319.619,Z 466.786,A -85,B 0,C 180,E1 -16588.571,E2 -16588.571} C_VEL
LIN {X 0,Y 319.78,Z 465.206,A -85,B 0,C 180,E1 -16588.914,E2 -16588.914} C_VEL
LIN {X 0,Y 318.647,Z 458.086,A -85,B 0,C 180,E1 -16591.03,E2 -16591.03} C_VEL
LIN {X 0,Y 317.352,Z 453.286,A -85,B 0,C 180,E1 -16592.695,E2 -16592.695} C_VEL
LIN {X 0,Y 316.145,Z 451.169,A -85,B 0,C 180,E1 -16593.763,E2 -16593.763} C_VEL
LIN {X 0,Y 313.245,Z 448.231,A -85,B 0,C 180,E1 -16596.127,E2 -16596.127} C_VEL
LIN {X 0,Y 311.496,Z 447.01,A -85,B 0,C 180,E1 -16597.844,E2 -16597.844} C_VEL
LIN {X 0,Y 309.923,Z 446.782,A -85,B 0,C 180,E1 -16599.554,E2 -16599.554} C_VEL
LIN {X 0,Y 308.948,Z 446.864,A -85,B 0,C 180,E1 -16601.348,E2 -16601.348} C_VEL
LIN {X 0,Y 308.284,Z 447.908,A -85,B 0,C 180,E1 -16603.153,E2 -16603.153} C_VEL
LIN {X 0,Y 308.044,Z 451.548,A -85,B 0,C 180,E1 -16605.995,E2 -16605.995} C_VEL
LIN {X 0,Y 308.476,Z 454.383,A -85,B 0,C 180,E1 -16607.599,E2 -16607.599} C_VEL
LIN {X 0,Y 308.458,Z 456.671,A -85,B 0,C 180,E1 -16608.327,E2 -16608.327} C_VEL
LIN {X 0,Y 308.691,Z 465.397,A -85,B 0,C 180,E1 -16610.722,E2 -16610.722} C_VEL
LIN {X 0,Y 309.173,Z 472.6,A -85,B 0,C 180,E1 -16612.437,E2 -16612.437} C_VEL
LIN {X 0,Y 309.759,Z 482.28,A -85,B 0,C 180,E1 -16614.44,E2 -16614.44} C_VEL
LIN {X 0,Y 310.019,Z 493.277,A -85,B 0,C 180,E1 -16616.417,E2 -16616.417} C_VEL
LIN {X 0,Y 309.831,Z 503.443,A -85,B 0,C 180,E1 -16618.105,E2 -16618.105} C_VEL
LIN {X 0,Y 308.639,Z 516.309,A -85,B 0,C 180,E1 -16620.107,E2 -16620.107} C_VEL
LIN {X 0,Y 306.329,Z 528.344,A -85,B 0,C 180,E1 -16621.943,E2 -16621.943} C_VEL
LIN {X 0,Y 303.548,Z 540.127,A -85,B 0,C 180,E1 -16623.901,E2 -16623.901} C_VEL
LIN {X 0,Y 301.591,Z 547.262,A -85,B 0,C 180,E1 -16625.199,E2 -16625.199} C_VEL
LIN {X 0,Y 298.46,Z 556.944,A -85,B 0,C 180,E1 -16627.135,E2 -16627.135} C_VEL
LIN {X 0,Y 295.17,Z 567.959,A -85,B 0,C 180,E1 -16629.802,E2 -16629.802} C_VEL
LIN {X 0,Y 292.769,Z 577.19,A -85,B 0,C 180,E1 -16632.537,E2 -16632.537} C_VEL
LIN {X 0,Y 291.138,Z 584.892,A -85,B 0,C 180,E1 -16635.348,E2 -16635.348} C_VEL
LIN {X 0,Y 290.389,Z 590.943,A -85,B 0,C 180,E1 -16638.127,E2 -16638.127} C_VEL
LIN {X 0,Y 290.223,Z 594.575,A -85,B 0,C 180,E1 -16640.239,E2 -16640.239} C_VEL
LIN {X 0,Y 290.464,Z 598.218,A -85,B 0,C 180,E1 -16643.05,E2 -16643.05} C_VEL
LIN {X 0,Y 290.724,Z 599.513,A -85,B 0,C 180,E1 -16644.45,E2 -16644.45} C_VEL
LIN {X 0,Y 291.126,Z 601.004,A -85,B 0,C 180,E1 -16647.231,E2 -16647.231} C_VEL
LIN {X 0,Y 291.478,Z 601.496,A -85,B 0,C 180,E1 -16648.617,E2 -16648.617} C_VEL
LIN {X 0,Y 291.727,Z 601.571,A -85,B 0,C 180,E1 -16649.999,E2 -16649.999} C_VEL
LIN {X 0,Y 291.507,Z 601.176,A -85,B 0,C 180,E1 -16651.38,E2 -16651.38} C_VEL
LIN {X 0,Y 291.278,Z 600.344,A -85,B 0,C 180,E1 -16652.764,E2 -16652.764} C_VEL
LIN {X 0,Y 291.104,Z 599.055,A -85,B 0,C 180,E1 -16654.152,E2 -16654.152} C_VEL
LIN {X 0,Y 290.947,Z 596.317,A -85,B 0,C 180,E1 -16656.239,E2 -16656.239} C_VEL
LIN {X 0,Y 290.727,Z 592.481,A -85,B 0,C 180,E1 -16658.338,E2 -16658.338} C_VEL
LIN {X 0,Y 290.69,Z 587.473,A -85,B 0,C 180,E1 -16660.445,E2 -16660.445} C_VEL
LIN {X 0,Y 290.919,Z 581.158,A -85,B 0,C 180,E1 -16662.556,E2 -16662.556} C_VEL
LIN {X 0,Y 291.524,Z 573.341,A -85,B 0,C 180,E1 -16664.661,E2 -16664.661} C_VEL
LIN {X 0,Y 292.273,Z 565.328,A -85,B 0,C 180,E1 -16666.414,E2 -16666.414} C_VEL
LIN {X 0,Y 294.263,Z 549.43,A -85,B 0,C 180,E1 -16669.351,E2 -16669.351} C_VEL
LIN {X 0,Y 295.716,Z 538.093,A -85,B 0,C 180,E1 -16671.065,E2 -16671.065} C_VEL
LIN {X 0,Y 296.328,Z 531.478,A -85,B 0,C 180,E1 -16671.932,E2 -16671.932} C_VEL
LIN {X 0,Y 295.49,Z 518.068,A -85,B 0,C 180,E1 -16673.475,E2 -16673.475} C_VEL
LIN {X 0,Y 294.363,Z 503.31,A -85,B 0,C 180,E1 -16674.871,E2 -16674.871} C_VEL
LIN {X 0,Y 293.081,Z 487.804,A -85,B 0,C 180,E1 -16676.038,E2 -16676.038} C_VEL
LIN {X 0,Y 291.758,Z 471.641,A -85,B 0,C 180,E1 -16676.967,E2 -16676.967} C_VEL
LIN {X 0,Y 292.831,Z 461.852,A -85,B 0,C 180,E1 -16681.062,E2 -16681.062} C_VEL
LIN {X 0,Y 294.123,Z 452.555,A -85,B 0,C 180,E1 -16684.991,E2 -16684.991} C_VEL
LIN {X 0,Y 295.676,Z 443.045,A -85,B 0,C 180,E1 -16689.038,E2 -16689.038} C_VEL
LIN {X 0,Y 296.282,Z 438.41,A -85,B 0,C 180,E1 -16691.052,E2 -16691.052} C_VEL
LIN {X 0,Y 295.554,Z 433.819,A -85,B 0,C 180,E1 -16693.169,E2 -16693.169} C_VEL
LIN {X 0,Y 293.934,Z 425.72,A -85,B 0,C 180,E1 -16697.044,E2 -16697.044} C_VEL
LIN {X 0,Y 292.224,Z 417.275,A -85,B 0,C 180,E1 -16701.296,E2 -16701.296} C_VEL
LIN {X 0,Y 291.397,Z 412.814,A -85,B 0,C 180,E1 -16703.672,E2 -16703.672} C_VEL
LIN {X 0,Y 291.363,Z 412.815,A -85,B 0,C 180,E1 -16707.95,E2 -16707.95} C_VEL
LIN {X 0,Y 291.376,Z 412.814,A -85,B 0,C 180,E1 -16711.158,E2 -16711.158} C_VEL
LIN {X 0,Y 291.411,Z 412.808,A -85,B 0,C 180,E1 -16714.272,E2 -16714.272} C_VEL
LIN {X 0,Y 291.371,Z 412.816,A -85,B 0,C 180,E1 -16717.299,E2 -16717.299} C_VEL
LIN {X 0,Y 291.448,Z 412.801,A -85,B 0,C 180,E1 -16720.27,E2 -16720.27} C_VEL
LIN {X 0,Y 291.545,Z 412.792,A -85,B 0,C 180,E1 -16724.623,E2 -16724.623} C_VEL
LIN {X 0,Y 291.529,Z 412.796,A -85,B 0,C 180,E1 -16728.881,E2 -16728.881} C_VEL
LIN {X 0,Y 291.699,Z 412.773,A -85,B 0,C 180,E1 -16731.689,E2 -16731.689} C_VEL
LIN {X 0,Y 291.622,Z 412.782,A -85,B 0,C 180,E1 -16734.468,E2 -16734.468} C_VEL
LIN {X 0,Y 291.884,Z 412.752,A -85,B 0,C 180,E1 -16738.621,E2 -16738.621} C_VEL
LIN {X 0,Y 291.884,Z 412.749,A -85,B 0,C 180,E1 -16741.38,E2 -16741.38} C_VEL
LIN {X 0,Y 291.737,Z 412.762,A -85,B 0,C 180,E1 -16746.919,E2 -16746.919} C_VEL
LIN {X 0,Y 291.62,Z 412.77,A -85,B 0,C 180,E1 -16749.713,E2 -16749.713} C_VEL
LIN {X 0,Y 291.514,Z 412.796,A -85,B 0,C 180,E1 -16753.951,E2 -16753.951} C_VEL
LIN {X 0,Y 291.478,Z 412.8,A -85,B 0,C 180,E1 -16756.819,E2 -16756.819} C_VEL
LIN {X 0,Y 291.442,Z 412.805,A -85,B 0,C 180,E1 -16759.876,E2 -16759.876} C_VEL
LIN {X 0,Y 291.392,Z 412.811,A -85,B 0,C 180,E1 -16764.206,E2 -16764.206} C_VEL
LIN {X 0,Y 291.415,Z 412.803,A -85,B 0,C 180,E1 -16767.273,E2 -16767.273} C_VEL
LIN {X 0,Y 291.33,Z 412.806,A -85,B 0,C 180,E1 -16770.438,E2 -16770.438} C_VEL
LIN {X 0,Y 291.338,Z 412.816,A -85,B 0,C 180,E1 -16773.7,E2 -16773.7} C_VEL
LIN {X 0,Y 291.37,Z 412.805,A -85,B 0,C 180,E1 -16777.256,E2 -16777.256} C_VEL
LIN {X 0,Y 291.327,Z 412.82,A -85,B 0,C 180,E1 -16780.644,E2 -16780.644} C_VEL
LIN {X 0,Y 291.309,Z 412.818,A -85,B 0,C 180,E1 -16784.399,E2 -16784.399} C_VEL
LIN {X 0,Y 291.352,Z 412.82,A -85,B 0,C 180,E1 -16788.4,E2 -16788.4} C_VEL
LIN {X 0,Y 291.377,Z 412.81,A -85,B 0,C 180,E1 -16791.165,E2 -16791.165} C_VEL
LIN {X 0,Y 291.384,Z 412.815,A -85,B 0,C 180,E1 -16794.632,E2 -16794.632} C_VEL
LIN {X 0,Y 291.371,Z 412.815,A -85,B 0,C 180,E1 -16797.953,E2 -16797.953} C_VEL
LIN {X 0,Y 291.38,Z 412.813,A -85,B 0,C 180,E1 -16801.16,E2 -16801.16} C_VEL
LIN {X 0,Y 291.416,Z 412.812,A -85,B 0,C 180,E1 -16804.274,E2 -16804.274} C_VEL
LIN {X 0,Y 291.392,Z 412.817,A -85,B 0,C 180,E1 -16808.049,E2 -16808.049} C_VEL
LIN {X 0,Y 291.397,Z 412.816,A -85,B 0,C 180,E1 -16808.746,E2 -16808.746} C_VEL
LIN {X 0,Y 292.428,Z 415.701,A -85,B 0,C 180,E1 -16808.936,E2 -16808.936} C_VEL
LIN {X 0,Y 297.51,Z 427.765,A -85,B 0,C 180,E1 -16809.915,E2 -16809.915} C_VEL
LIN {X 0,Y 301.073,Z 438.454,A -85,B 0,C 180,E1 -16810.927,E2 -16810.927} C_VEL
LIN {X 0,Y 301.849,Z 442.345,A -85,B 0,C 180,E1 -16811.311,E2 -16811.311} C_VEL
LIN {X 0,Y 300.987,Z 453.519,A -85,B 0,C 180,E1 -16812.331,E2 -16812.331} C_VEL
LIN {X 0,Y 299.81,Z 464.853,A -85,B 0,C 180,E1 -16813.664,E2 -16813.664} C_VEL
LIN {X 0,Y 298.373,Z 475.666,A -85,B 0,C 180,E1 -16815.269,E2 -16815.269} C_VEL
LIN {X 0,Y 296.943,Z 485.03,A -85,B 0,C 180,E1 -16817.008,E2 -16817.008} C_VEL
LIN {X 0,Y 295.569,Z 493.685,A -85,B 0,C 180,E1 -16819.036,E2 -16819.036} C_VEL
LIN {X 0,Y 294.366,Z 500.669,A -85,B 0,C 180,E1 -16821.074,E2 -16821.074} C_VEL
LIN {X 0,Y 293.576,Z 506.223,A -85,B 0,C 180,E1 -16823.127,E2 -16823.127} C_VEL
LIN {X 0,Y 292.788,Z 510.602,A -85,B 0,C 180,E1 -16825.182,E2 -16825.182} C_VEL
LIN {X 0,Y 292.128,Z 513.931,A -85,B 0,C 180,E1 -16827.244,E2 -16827.244} C_VEL
LIN {X 0,Y 291.767,Z 516.825,A -85,B 0,C 180,E1 -16830.001,E2 -16830.001} C_VEL
LIN {X 0,Y 291.745,Z 517.694,A -85,B 0,C 180,E1 -16831.382,E2 -16831.382} C_VEL
LIN {X 0,Y 291.634,Z 518.181,A -85,B 0,C 180,E1 -16832.764,E2 -16832.764} C_VEL
LIN {X 0,Y 291.523,Z 518.278,A -85,B 0,C 180,E1 -16834.149,E2 -16834.149} C_VEL
LIN {X 0,Y 292.117,Z 517.277,A -85,B 0,C 180,E1 -16836.911,E2 -16836.911} C_VEL
LIN {X 0,Y 292.598,Z 516.154,A -85,B 0,C 180,E1 -16838.287,E2 -16838.287} C_VEL
LIN {X 0,Y 293.362,Z 513.088,A -85,B 0,C 180,E1 -16840.816,E2 -16840.816} C_VEL
LIN {X 0,Y 294.406,Z 509.006,A -85,B 0,C 180,E1 -16843.109,E2 -16843.109} C_VEL
LIN {X 0,Y 295.411,Z 504.167,A -85,B 0,C 180,E1 -16845.172,E2 -16845.172} C_VEL
LIN {X 0,Y 296.655,Z 498.014,A -85,B 0,C 180,E1 -16847.227,E2 -16847.227} C_VEL
LIN {X 0,Y 298.245,Z 490.277,A -85,B 0,C 180,E1 -16849.264,E2 -16849.264} C_VEL
LIN {X 0,Y 299.801,Z 482.344,A -85,B 0,C 180,E1 -16850.948,E2 -16850.948} C_VEL
LIN {X 0,Y 301.342,Z 472.654,A -85,B 0,C 180,E1 -16852.634,E2 -16852.634} C_VEL
LIN {X 0,Y 302.8,Z 461.667,A -85,B 0,C 180,E1 -16854.148,E2 -16854.148} C_VEL
LIN {X 0,Y 304.044,Z 450.139,A -85,B 0,C 180,E1 -16855.4,E2 -16855.4} C_VEL
LIN {X 0,Y 304.481,Z 445.474,A -85,B 0,C 180,E1 -16855.815,E2 -16855.815} C_VEL
LIN {X 0,Y 301.091,Z 434.94,A -85,B 0,C 180,E1 -16857.017,E2 -16857.017} C_VEL
LIN {X 0,Y 296.424,Z 423.748,A -85,B 0,C 180,E1 -16858.156,E2 -16858.156} C_VEL
LIN {X 0,Y 292.256,Z 415.319,A -85,B 0,C 180,E1 -16858.933,E2 -16858.933} C_VEL
LIN {X 0,Y 291.426,Z 412.81,A -85,B 0,C 180,E1 -16859.135,E2 -16859.135} C_VEL
LIN {X 0,Y 291.35,Z 412.821,A -85,B 0,C 180,E1 -16862.404,E2 -16862.404} C_VEL
LIN {X 0,Y 291.367,Z 412.82,A -85,B 0,C 180,E1 -16865.374,E2 -16865.374} C_VEL
LIN {X 0,Y 291.353,Z 412.801,A -85,B 0,C 180,E1 -16868.843,E2 -16868.843} C_VEL
LIN {X 0,Y 291.325,Z 412.817,A -85,B 0,C 180,E1 -16872.493,E2 -16872.493} C_VEL
LIN {X 0,Y 291.315,Z 412.819,A -85,B 0,C 180,E1 -16876.367,E2 -16876.367} C_VEL
LIN {X 0,Y 291.384,Z 412.78,A -85,B 0,C 180,E1 -16880.519,E2 -16880.519} C_VEL
LIN {X 0,Y 291.41,Z 412.789,A -85,B 0,C 180,E1 -16882.919,E2 -16882.919} C_VEL
LIN {X 0,Y 291.35,Z 412.816,A -85,B 0,C 180,E1 -16886.302,E2 -16886.302} C_VEL
LIN {X 0,Y 291.389,Z 412.764,A -85,B 0,C 180,E1 -16890.262,E2 -16890.262} C_VEL
LIN {X 0,Y 291.419,Z 412.806,A -85,B 0,C 180,E1 -16894.272,E2 -16894.272} C_VEL
LIN {X 0,Y 291.457,Z 412.937,A -85,B 0,C 180,E1 -16896.18,E2 -16896.18} C_VEL
LIN {X 0,Y 295.092,Z 425.808,A -85,B 0,C 180,E1 -16897.508,E2 -16897.508} C_VEL
LIN {X 0,Y 298.674,Z 438.573,A -85,B 0,C 180,E1 -16899.064,E2 -16899.064} C_VEL
LIN {X 0,Y 299.123,Z 440.913,A -85,B 0,C 180,E1 -16899.364,E2 -16899.364} C_VEL
LIN {X 0,Y 297.723,Z 454.191,A -85,B 0,C 180,E1 -16901.059,E2 -16901.059} C_VEL
LIN {X 0,Y 296.374,Z 465.23,A -85,B 0,C 180,E1 -16902.757,E2 -16902.757} C_VEL
LIN {X 0,Y 295.053,Z 476.331,A -85,B 0,C 180,E1 -16904.81,E2 -16904.81} C_VEL
LIN {X 0,Y 294.302,Z 483.725,A -85,B 0,C 180,E1 -16906.415,E2 -16906.415} C_VEL
LIN {X 0,Y 293.197,Z 487.467,A -85,B 0,C 180,E1 -16907.282,E2 -16907.282} C_VEL
LIN {X 0,Y 289.693,Z 493.306,A -85,B 0,C 180,E1 -16908.704,E2 -16908.704} C_VEL
LIN {X 0,Y 286.318,Z 498.696,A -85,B 0,C 180,E1 -16910.222,E2 -16910.222} C_VEL
LIN {X 0,Y 285.435,Z 501.719,A -85,B 0,C 180,E1 -16911.224,E2 -16911.224} C_VEL
LIN {X 0,Y 284.949,Z 507.902,A -85,B 0,C 180,E1 -16913.627,E2 -16913.627} C_VEL
LIN {X 0,Y 284.394,Z 512.404,A -85,B 0,C 180,E1 -16915.748,E2 -16915.748} C_VEL
LIN {X 0,Y 284.703,Z 516.974,A -85,B 0,C 180,E1 -16918.585,E2 -16918.585} C_VEL
LIN {X 0,Y 284.818,Z 520.204,A -85,B 0,C 180,E1 -16921.414,E2 -16921.414} C_VEL
LIN {X 0,Y 285.434,Z 522.099,A -85,B 0,C 180,E1 -16924.236,E2 -16924.236} C_VEL
LIN {X 0,Y 286.41,Z 522.696,A -85,B 0,C 180,E1 -16927.047,E2 -16927.047} C_VEL
LIN {X 0,Y 287.867,Z 522.009,A -85,B 0,C 180,E1 -16929.84,E2 -16929.84} C_VEL
LIN {X 0,Y 289.838,Z 520.033,A -85,B 0,C 180,E1 -16932.605,E2 -16932.605} C_VEL
LIN {X 0,Y 292.146,Z 516.759,A -85,B 0,C 180,E1 -16935.344,E2 -16935.344} C_VEL
LIN {X 0,Y 295.078,Z 512.069,A -85,B 0,C 180,E1 -16938.036,E2 -16938.036} C_VEL
LIN {X 0,Y 298.516,Z 505.923,A -85,B 0,C 180,E1 -16940.68,E2 -16940.68} C_VEL
LIN {X 0,Y 302.552,Z 498.108,A -85,B 0,C 180,E1 -16943.259,E2 -16943.259} C_VEL
LIN {X 0,Y 307.063,Z 488.35,A -85,B 0,C 180,E1 -16945.777,E2 -16945.777} C_VEL
LIN {X 0,Y 310.868,Z 479.421,A -85,B 0,C 180,E1 -16947.643,E2 -16947.643} C_VEL
LIN {X 0,Y 314.698,Z 469.341,A -85,B 0,C 180,E1 -16949.427,E2 -16949.427} C_VEL
LIN {X 0,Y 314.092,Z 463.513,A -85,B 0,C 180,E1 -16951.248,E2 -16951.248} C_VEL
LIN {X 0,Y 313.076,Z 458.596,A -85,B 0,C 180,E1 -16953.063,E2 -16953.063} C_VEL
LIN {X 0,Y 311.821,Z 456.486,A -85,B 0,C 180,E1 -16954.295,E2 -16954.295} C_VEL
LIN {X 0,Y 309.844,Z 454.448,A -85,B 0,C 180,E1 -16956.138,E2 -16956.138} C_VEL
LIN {X 0,Y 308.106,Z 453.3,A -85,B 0,C 180,E1 -16958.016,E2 -16958.016} C_VEL
LIN {X 0,Y 306.156,Z 453.235,A -85,B 0,C 180,E1 -16960.751,E2 -16960.751} C_VEL
LIN {X 0,Y 305.446,Z 454.069,A -85,B 0,C 180,E1 -16962.583,E2 -16962.583} C_VEL
LIN {X 0,Y 305.032,Z 455.972,A -85,B 0,C 180,E1 -16964.417,E2 -16964.417} C_VEL
LIN {X 0,Y 305.174,Z 459.504,A -85,B 0,C 180,E1 -16966.745,E2 -16966.745} C_VEL
LIN {X 0,Y 305.264,Z 461.057,A -85,B 0,C 180,E1 -16967.453,E2 -16967.453} C_VEL
LIN {X 0,Y 304.889,Z 470.519,A -85,B 0,C 180,E1 -16970.135,E2 -16970.135} C_VEL
LIN {X 0,Y 305.006,Z 478.512,A -85,B 0,C 180,E1 -16972.093,E2 -16972.093} C_VEL
LIN {X 0,Y 305.122,Z 487.996,A -85,B 0,C 180,E1 -16974.118,E2 -16974.118} C_VEL
LIN {X 0,Y 304.801,Z 500.241,A -85,B 0,C 180,E1 -16976.399,E2 -16976.399} C_VEL
LIN {X 0,Y 303.67,Z 512.481,A -85,B 0,C 180,E1 -16978.481,E2 -16978.481} C_VEL
LIN {X 0,Y 301.893,Z 523.187,A -85,B 0,C 180,E1 -16980.233,E2 -16980.233} C_VEL
LIN {X 0,Y 298.159,Z 537.563,A -85,B 0,C 180,E1 -16982.635,E2 -16982.635} C_VEL
LIN {X 0,Y 295.807,Z 546.317,A -85,B 0,C 180,E1 -16984.303,E2 -16984.303} C_VEL
LIN {X 0,Y 292.415,Z 555.84,A -85,B 0,C 180,E1 -16986.259,E2 -16986.259} C_VEL
LIN {X 0,Y 288.863,Z 566.72,A -85,B 0,C 180,E1 -16988.968,E2 -16988.968} C_VEL
LIN {X 0,Y 286.177,Z 575.861,A -85,B 0,C 180,E1 -16991.751,E2 -16991.751} C_VEL
LIN {X 0,Y 284.457,Z 583.166,A -85,B 0,C 180,E1 -16994.485,E2 -16994.485} C_VEL
LIN {X 0,Y 283.51,Z 588.836,A -85,B 0,C 180,E1 -16997.107,E2 -16997.107} C_VEL
LIN {X 0,Y 283.139,Z 593.709,A -85,B 0,C 180,E1 -16999.992,E2 -16999.992} C_VEL
LIN {X 0,Y 283.396,Z 597.217,A -85,B 0,C 180,E1 -17002.876,E2 -17002.876} C_VEL
LIN {X 0,Y 283.663,Z 598.449,A -85,B 0,C 180,E1 -17004.311,E2 -17004.311} C_VEL
LIN {X 0,Y 284.073,Z 599.984,A -85,B 0,C 180,E1 -17007.162,E2 -17007.162} C_VEL
LIN {X 0,Y 284.435,Z 600.486,A -85,B 0,C 180,E1 -17008.583,E2 -17008.583} C_VEL
LIN {X 0,Y 284.698,Z 600.563,A -85,B 0,C 180,E1 -17009.998,E2 -17009.998} C_VEL
LIN {X 0,Y 284.471,Z 600.159,A -85,B 0,C 180,E1 -17011.414,E2 -17011.414} C_VEL
LIN {X 0,Y 284.22,Z 599.309,A -85,B 0,C 180,E1 -17012.833,E2 -17012.833} C_VEL
LIN {X 0,Y 284.054,Z 598.012,A -85,B 0,C 180,E1 -17014.255,E2 -17014.255} C_VEL
LIN {X 0,Y 283.858,Z 595.249,A -85,B 0,C 180,E1 -17016.395,E2 -17016.395} C_VEL
LIN {X 0,Y 283.65,Z 591.394,A -85,B 0,C 180,E1 -17018.548,E2 -17018.548} C_VEL
LIN {X 0,Y 283.624,Z 586.364,A -85,B 0,C 180,E1 -17020.709,E2 -17020.709} C_VEL
LIN {X 0,Y 283.921,Z 580.032,A -85,B 0,C 180,E1 -17022.871,E2 -17022.871} C_VEL
LIN {X 0,Y 284.561,Z 572.185,A -85,B 0,C 180,E1 -17025.028,E2 -17025.028} C_VEL
LIN {X 0,Y 285.392,Z 564.167,A -85,B 0,C 180,E1 -17026.817,E2 -17026.817} C_VEL
LIN {X 0,Y 286.53,Z 554.389,A -85,B 0,C 180,E1 -17028.592,E2 -17028.592} C_VEL
LIN {X 0,Y 288.683,Z 537.567,A -85,B 0,C 180,E1 -17031.229,E2 -17031.229} C_VEL
LIN {X 0,Y 289.252,Z 531.711,A -85,B 0,C 180,E1 -17032.026,E2 -17032.026} C_VEL
LIN {X 0,Y 288.539,Z 519.558,A -85,B 0,C 180,E1 -17033.504,E2 -17033.504} C_VEL
LIN {X 0,Y 287.518,Z 505.94,A -85,B 0,C 180,E1 -17034.89,E2 -17034.89} C_VEL
LIN {X 0,Y 286.322,Z 490.52,A -85,B 0,C 180,E1 -17036.142,E2 -17036.142} C_VEL
LIN {X 0,Y 285.004,Z 474.635,A -85,B 0,C 180,E1 -17037.132,E2 -17037.132} C_VEL
LIN {X 0,Y 284.736,Z 470.735,A -85,B 0,C 180,E1 -17037.372,E2 -17037.372} C_VEL
LIN {X 0,Y 285.753,Z 462.083,A -85,B 0,C 180,E1 -17041.095,E2 -17041.095} C_VEL
LIN {X 0,Y 287.062,Z 452.794,A -85,B 0,C 180,E1 -17045.121,E2 -17045.121} C_VEL
LIN {X 0,Y 288.685,Z 443.36,A -85,B 0,C 180,E1 -17049.267,E2 -17049.267} C_VEL
LIN {X 0,Y 289.229,Z 439.184,A -85,B 0,C 180,E1 -17051.126,E2 -17051.126} C_VEL
LIN {X 0,Y 288.573,Z 435.058,A -85,B 0,C 180,E1 -17053.061,E2 -17053.061} C_VEL
LIN {X 0,Y 286.833,Z 426.387,A -85,B 0,C 180,E1 -17057.309,E2 -17057.309} C_VEL
LIN {X 0,Y 285.074,Z 417.416,A -85,B 0,C 180,E1 -17061.952,E2 -17061.952} C_VEL
LIN {X 0,Y 284.348,Z 413.69,A -85,B 0,C 180,E1 -17064.053,E2 -17064.053} C_VEL
LIN {X 0,Y 284.299,Z 413.697,A -85,B 0,C 180,E1 -17067.189,E2 -17067.189} C_VEL
LIN {X 0,Y 284.35,Z 413.687,A -85,B 0,C 180,E1 -17070.375,E2 -17070.375} C_VEL
LIN {X 0,Y 284.371,Z 413.686,A -85,B 0,C 180,E1 -17073.586,E2 -17073.586} C_VEL
LIN {X 0,Y 284.357,Z 413.688,A -85,B 0,C 180,E1 -17076.706,E2 -17076.706} C_VEL
LIN {X 0,Y 284.394,Z 413.686,A -85,B 0,C 180,E1 -17081.261,E2 -17081.261} C_VEL
LIN {X 0,Y 284.482,Z 413.67,A -85,B 0,C 180,E1 -17084.459,E2 -17084.459} C_VEL
LIN {X 0,Y 284.48,Z 413.673,A -85,B 0,C 180,E1 -17088.601,E2 -17088.601} C_VEL
LIN {X 0,Y 284.649,Z 413.652,A -85,B 0,C 180,E1 -17091.481,E2 -17091.481} C_VEL
LIN {X 0,Y 284.593,Z 413.657,A -85,B 0,C 180,E1 -17094.331,E2 -17094.331} C_VEL
LIN {X 0,Y 284.85,Z 413.628,A -85,B 0,C 180,E1 -17098.587,E2 -17098.587} C_VEL
LIN {X 0,Y 284.85,Z 413.625,A -85,B 0,C 180,E1 -17101.414,E2 -17101.414} C_VEL
LIN {X 0,Y 284.689,Z 413.637,A -85,B 0,C 180,E1 -17107.091,E2 -17107.091} C_VEL
LIN {X 0,Y 284.558,Z 413.649,A -85,B 0,C 180,E1 -17109.956,E2 -17109.956} C_VEL
LIN {X 0,Y 284.473,Z 413.674,A -85,B 0,C 180,E1 -17114.304,E2 -17114.304} C_VEL
LIN {X 0,Y 284.417,Z 413.678,A -85,B 0,C 180,E1 -17117.249,E2 -17117.249} C_VEL
LIN {X 0,Y 284.37,Z 413.687,A -85,B 0,C 180,E1 -17120.243,E2 -17120.243} C_VEL
LIN {X 0,Y 284.361,Z 413.686,A -85,B 0,C 180,E1 -17123.877,E2 -17123.877} C_VEL
LIN {X 0,Y 284.389,Z 413.679,A -85,B 0,C 180,E1 -17127.175,E2 -17127.175} C_VEL
LIN {X 0,Y 284.288,Z 413.69,A -85,B 0,C 180,E1 -17131.276,E2 -17131.276} C_VEL
LIN {X 0,Y 284.334,Z 413.688,A -85,B 0,C 180,E1 -17135.35,E2 -17135.35} C_VEL
LIN {X 0,Y 284.306,Z 413.684,A -85,B 0,C 180,E1 -17138.171,E2 -17138.171} C_VEL
LIN {X 0,Y 284.264,Z 413.7,A -85,B 0,C 180,E1 -17142.126,E2 -17142.126} C_VEL
LIN {X 0,Y 284.281,Z 413.691,A -85,B 0,C 180,E1 -17146.197,E2 -17146.197} C_VEL
LIN {X 0,Y 284.348,Z 413.689,A -85,B 0,C 180,E1 -17150.015,E2 -17150.015} C_VEL
LIN {X 0,Y 284.353,Z 413.688,A -85,B 0,C 180,E1 -17153.619,E2 -17153.619} C_VEL
LIN {X 0,Y 284.306,Z 413.694,A -85,B 0,C 180,E1 -17157.191,E2 -17157.191} C_VEL
LIN {X 0,Y 284.357,Z 413.689,A -85,B 0,C 180,E1 -17160.378,E2 -17160.378} C_VEL
LIN {X 0,Y 284.377,Z 413.687,A -85,B 0,C 180,E1 -17163.589,E2 -17163.589} C_VEL
LIN {X 0,Y 284.355,Z 413.693,A -85,B 0,C 180,E1 -17167.477,E2 -17167.477} C_VEL
LIN {X 0,Y 284.361,Z 413.693,A -85,B 0,C 180,E1 -17168.146,E2 -17168.146} C_VEL
LIN {X 0,Y 285.372,Z 416.597,A -85,B 0,C 180,E1 -17168.336,E2 -17168.336} C_VEL
LIN {X 0,Y 290.706,Z 428.917,A -85,B 0,C 180,E1 -17169.386,E2 -17169.386} C_VEL
LIN {X 0,Y 294.394,Z 440.027,A -85,B 0,C 180,E1 -17170.477,E2 -17170.477} C_VEL
LIN {X 0,Y 295.228,Z 443.786,A -85,B 0,C 180,E1 -17170.872,E2 -17170.872} C_VEL
LIN {X 0,Y 294.346,Z 454.9,A -85,B 0,C 180,E1 -17171.919,E2 -17171.919} C_VEL
LIN {X 0,Y 293.119,Z 466.137,A -85,B 0,C 180,E1 -17173.28,E2 -17173.28} C_VEL
LIN {X 0,Y 291.665,Z 476.562,A -85,B 0,C 180,E1 -17174.863,E2 -17174.863} C_VEL
LIN {X 0,Y 290.123,Z 486.214,A -85,B 0,C 180,E1 -17176.697,E2 -17176.697} C_VEL
LIN {X 0,Y 288.695,Z 494.841,A -85,B 0,C 180,E1 -17178.771,E2 -17178.771} C_VEL
LIN {X 0,Y 287.438,Z 501.8,A -85,B 0,C 180,E1 -17180.857,E2 -17180.857} C_VEL
LIN {X 0,Y 286.618,Z 507.322,A -85,B 0,C 180,E1 -17182.959,E2 -17182.959} C_VEL
LIN {X 0,Y 285.794,Z 511.679,A -85,B 0,C 180,E1 -17185.064,E2 -17185.064} C_VEL
LIN {X 0,Y 285.112,Z 514.99,A -85,B 0,C 180,E1 -17187.176,E2 -17187.176} C_VEL
LIN {X 0,Y 284.742,Z 517.861,A -85,B 0,C 180,E1 -17190.002,E2 -17190.002} C_VEL
LIN {X 0,Y 284.723,Z 518.721,A -85,B 0,C 180,E1 -17191.416,E2 -17191.416} C_VEL
LIN {X 0,Y 284.61,Z 519.191,A -85,B 0,C 180,E1 -17192.832,E2 -17192.832} C_VEL
LIN {X 0,Y 284.506,Z 519.279,A -85,B 0,C 180,E1 -17194.251,E2 -17194.251} C_VEL
LIN {X 0,Y 285.137,Z 518.255,A -85,B 0,C 180,E1 -17197.081,E2 -17197.081} C_VEL
LIN {X 0,Y 285.641,Z 517.115,A -85,B 0,C 180,E1 -17198.491,E2 -17198.491} C_VEL
LIN {X 0,Y 286.548,Z 513.688,A -85,B 0,C 180,E1 -17201.317,E2 -17201.317} C_VEL
LIN {X 0,Y 287.556,Z 509.926,A -85,B 0,C 180,E1 -17203.427,E2 -17203.427} C_VEL
LIN {X 0,Y 288.618,Z 505.061,A -85,B 0,C 180,E1 -17205.538,E2 -17205.538} C_VEL
LIN {X 0,Y 289.929,Z 498.872,A -85,B 0,C 180,E1 -17207.64,E2 -17207.64} C_VEL
LIN {X 0,Y 291.611,Z 491.103,A -85,B 0,C 180,E1 -17209.72,E2 -17209.72} C_VEL
LIN {X 0,Y 293.22,Z 483.136,A -85,B 0,C 180,E1 -17211.441,E2 -17211.441} C_VEL
LIN {X 0,Y 294.843,Z 473.379,A -85,B 0,C 180,E1 -17213.161,E2 -17213.161} C_VEL
LIN {X 0,Y 296.369,Z 462.327,A -85,B 0,C 180,E1 -17214.707,E2 -17214.707} C_VEL
LIN {X 0,Y 297.605,Z 451.268,A -85,B 0,C 180,E1 -17215.929,E2 -17215.929} C_VEL
LIN {X 0,Y 297.955,Z 447.053,A -85,B 0,C 180,E1 -17216.32,E2 -17216.32} C_VEL
LIN {X 0,Y 294.419,Z 436.418,A -85,B 0,C 180,E1 -17217.599,E2 -17217.599} C_VEL
LIN {X 0,Y 289.98,Z 425.686,A -85,B 0,C 180,E1 -17218.745,E2 -17218.745} C_VEL
LIN {X 0,Y 284.482,Z 414.47,A -85,B 0,C 180,E1 -17219.803,E2 -17219.803} C_VEL
LIN {X 0,Y 284.334,Z 413.695,A -85,B 0,C 180,E1 -17219.883,E2 -17219.883} C_VEL
LIN {X 0,Y 284.312,Z 413.698,A -85,B 0,C 180,E1 -17222.946,E2 -17222.946} C_VEL
LIN {X 0,Y 284.336,Z 413.691,A -85,B 0,C 180,E1 -17226.387,E2 -17226.387} C_VEL
LIN {X 0,Y 284.311,Z 413.691,A -85,B 0,C 180,E1 -17229.995,E2 -17229.995} C_VEL
LIN {X 0,Y 284.252,Z 413.704,A -85,B 0,C 180,E1 -17234.191,E2 -17234.191} C_VEL
LIN {X 0,Y 284.279,Z 413.697,A -85,B 0,C 180,E1 -17238.125,E2 -17238.125} C_VEL
LIN {X 0,Y 284.325,Z 413.661,A -85,B 0,C 180,E1 -17242.279,E2 -17242.279} C_VEL
LIN {X 0,Y 284.315,Z 413.695,A -85,B 0,C 180,E1 -17245.351,E2 -17245.351} C_VEL
LIN {X 0,Y 284.299,Z 413.66,A -85,B 0,C 180,E1 -17248.726,E2 -17248.726} C_VEL
LIN {X 0,Y 284.401,Z 413.661,A -85,B 0,C 180,E1 -17252.827,E2 -17252.827} C_VEL
LIN {X 0,Y 284.408,Z 413.685,A -85,B 0,C 180,E1 -17255.823,E2 -17255.823} C_VEL
LIN {X 0,Y 288.117,Z 426.987,A -85,B 0,C 180,E1 -17257.241,E2 -17257.241} C_VEL
LIN {X 0,Y 291.632,Z 439.551,A -85,B 0,C 180,E1 -17258.808,E2 -17258.808} C_VEL
LIN {X 0,Y 292.087,Z 442.695,A -85,B 0,C 180,E1 -17259.212,E2 -17259.212} C_VEL
LIN {X 0,Y 290.602,Z 456.262,A -85,B 0,C 180,E1 -17261.021,E2 -17261.021} C_VEL
LIN {X 0,Y 289.056,Z 468.692,A -85,B 0,C 180,E1 -17263.036,E2 -17263.036} C_VEL
LIN {X 0,Y 287.797,Z 479.452,A -85,B 0,C 180,E1 -17265.142,E2 -17265.142} C_VEL
LIN {X 0,Y 286.773,Z 488.473,A -85,B 0,C 180,E1 -17267.257,E2 -17267.257} C_VEL
LIN {X 0,Y 285.935,Z 496.415,A -85,B 0,C 180,E1 -17269.476,E2 -17269.476} C_VEL
LIN {X 0,Y 285.435,Z 501.719,A -85,B 0,C 180,E1 -17271.224,E2 -17271.224} C_VEL
LIN {X 0,Y 284.554,Z 504.604,A -85,B 0,C 180,E1 -17272.246,E2 -17272.246} C_VEL
LIN {X 0,Y 281.271,Z 508.992,A -85,B 0,C 180,E1 -17273.92,E2 -17273.92} C_VEL
LIN {X 0,Y 278.105,Z 512.981,A -85,B 0,C 180,E1 -17275.676,E2 -17275.676} C_VEL
LIN {X 0,Y 277.436,Z 515.059,A -85,B 0,C 180,E1 -17276.807,E2 -17276.807} C_VEL
LIN {X 0,Y 277.655,Z 517.756,A -85,B 0,C 180,E1 -17278.549,E2 -17278.549} C_VEL
LIN {X 0,Y 277.796,Z 521.158,A -85,B 0,C 180,E1 -17281.449,E2 -17281.449} C_VEL
LIN {X 0,Y 278.44,Z 523.229,A -85,B 0,C 180,E1 -17284.342,E2 -17284.342} C_VEL
LIN {X 0,Y 279.483,Z 524.007,A -85,B 0,C 180,E1 -17287.223,E2 -17287.223} C_VEL
LIN {X 0,Y 281.03,Z 523.508,A -85,B 0,C 180,E1 -17290.082,E2 -17290.082} C_VEL
LIN {X 0,Y 283.117,Z 521.737,A -85,B 0,C 180,E1 -17292.909,E2 -17292.909} C_VEL
LIN {X 0,Y 285.588,Z 518.717,A -85,B 0,C 180,E1 -17295.705,E2 -17295.705} C_VEL
LIN {X 0,Y 288.692,Z 514.318,A -85,B 0,C 180,E1 -17298.45,E2 -17298.45} C_VEL
LIN {X 0,Y 292.314,Z 508.451,A -85,B 0,C 180,E1 -17301.139,E2 -17301.139} C_VEL
LIN {X 0,Y 296.549,Z 500.993,A -85,B 0,C 180,E1 -17303.759,E2 -17303.759} C_VEL
LIN {X 0,Y 300.704,Z 492.998,A -85,B 0,C 180,E1 -17305.99,E2 -17305.99} C_VEL
LIN {X 0,Y 304.975,Z 483.918,A -85,B 0,C 180,E1 -17308.055,E2 -17308.055} C_VEL
LIN {X 0,Y 309.467,Z 473.542,A -85,B 0,C 180,E1 -17309.975,E2 -17309.975} C_VEL
LIN {X 0,Y 309.594,Z 470.923,A -85,B 0,C 180,E1 -17310.763,E2 -17310.763} C_VEL
LIN {X 0,Y 309.069,Z 465.528,A -85,B 0,C 180,E1 -17312.715,E2 -17312.715} C_VEL
LIN {X 0,Y 308.264,Z 462.931,A -85,B 0,C 180,E1 -17313.998,E2 -17313.998} C_VEL
LIN {X 0,Y 305.927,Z 460.33,A -85,B 0,C 180,E1 -17316.48,E2 -17316.48} C_VEL
LIN {X 0,Y 304.198,Z 459.468,A -85,B 0,C 180,E1 -17318.593,E2 -17318.593} C_VEL
LIN {X 0,Y 303.024,Z 459.535,A -85,B 0,C 180,E1 -17320.496,E2 -17320.496} C_VEL
LIN {X 0,Y 302.311,Z 460.357,A -85,B 0,C 180,E1 -17322.39,E2 -17322.39} C_VEL
LIN {X 0,Y 301.832,Z 462.377,A -85,B 0,C 180,E1 -17324.309,E2 -17324.309} C_VEL
LIN {X 0,Y 301.838,Z 465.158,A -85,B 0,C 180,E1 -17326.203,E2 -17326.203} C_VEL
LIN {X 0,Y 301.752,Z 467.124,A -85,B 0,C 180,E1 -17327.049,E2 -17327.049} C_VEL
LIN {X 0,Y 301.015,Z 475.218,A -85,B 0,C 180,E1 -17329.452,E2 -17329.452} C_VEL
LIN {X 0,Y 300.735,Z 482.256,A -85,B 0,C 180,E1 -17331.269,E2 -17331.269} C_VEL
LIN {X 0,Y 300.382,Z 491.95,A -85,B 0,C 180,E1 -17333.461,E2 -17333.461} C_VEL
LIN {X 0,Y 299.449,Z 504.836,A -85,B 0,C 180,E1 -17335.988,E2 -17335.988} C_VEL
LIN {X 0,Y 297.912,Z 515.708,A -85,B 0,C 180,E1 -17337.94,E2 -17337.94} C_VEL
LIN {X 0,Y 295.703,Z 526.221,A -85,B 0,C 180,E1 -17339.761,E2 -17339.761} C_VEL
LIN {X 0,Y 291.455,Z 540.535,A -85,B 0,C 180,E1 -17342.341,E2 -17342.341} C_VEL
LIN {X 0,Y 289.487,Z 547.182,A -85,B 0,C 180,E1 -17343.699,E2 -17343.699} C_VEL
LIN {X 0,Y 285.945,Z 556.297,A -85,B 0,C 180,E1 -17345.688,E2 -17345.688} C_VEL
LIN {X 0,Y 282.223,Z 566.821,A -85,B 0,C 180,E1 -17348.449,E2 -17348.449} C_VEL
LIN {X 0,Y 279.683,Z 574.608,A -85,B 0,C 180,E1 -17350.932,E2 -17350.932} C_VEL
LIN {X 0,Y 277.704,Z 582.109,A -85,B 0,C 180,E1 -17353.835,E2 -17353.835} C_VEL
LIN {X 0,Y 276.505,Z 588.175,A -85,B 0,C 180,E1 -17356.775,E2 -17356.775} C_VEL
LIN {X 0,Y 276.073,Z 592.868,A -85,B 0,C 180,E1 -17359.734,E2 -17359.734} C_VEL
LIN {X 0,Y 276.305,Z 596.267,A -85,B 0,C 180,E1 -17362.742,E2 -17362.742} C_VEL
LIN {X 0,Y 276.581,Z 597.388,A -85,B 0,C 180,E1 -17364.165,E2 -17364.165} C_VEL
LIN {X 0,Y 277.015,Z 598.986,A -85,B 0,C 180,E1 -17367.09,E2 -17367.09} C_VEL
LIN {X 0,Y 277.392,Z 599.482,A -85,B 0,C 180,E1 -17368.547,E2 -17368.547} C_VEL
LIN {X 0,Y 277.669,Z 599.554,A -85,B 0,C 180,E1 -17369.998,E2 -17369.998} C_VEL
LIN {X 0,Y 277.434,Z 599.142,A -85,B 0,C 180,E1 -17371.45,E2 -17371.45} C_VEL
LIN {X 0,Y 277.162,Z 598.273,A -85,B 0,C 180,E1 -17372.905,E2 -17372.905} C_VEL
LIN {X 0,Y 277.005,Z 596.969,A -85,B 0,C 180,E1 -17374.364,E2 -17374.364} C_VEL
LIN {X 0,Y 276.775,Z 594.182,A -85,B 0,C 180,E1 -17376.56,E2 -17376.56} C_VEL
LIN {X 0,Y 276.555,Z 590.304,A -85,B 0,C 180,E1 -17378.769,E2 -17378.769} C_VEL
LIN {X 0,Y 276.578,Z 585.256,A -85,B 0,C 180,E1 -17380.985,E2 -17380.985} C_VEL
LIN {X 0,Y 276.873,Z 578.896,A -85,B 0,C 180,E1 -17383.204,E2 -17383.204} C_VEL
LIN {X 0,Y 277.565,Z 571.382,A -85,B 0,C 180,E1 -17385.324,E2 -17385.324} C_VEL
LIN {X 0,Y 278.472,Z 562.967,A -85,B 0,C 180,E1 -17387.248,E2 -17387.248} C_VEL
LIN {X 0,Y 279.721,Z 553.164,A -85,B 0,C 180,E1 -17389.062,E2 -17389.062} C_VEL
LIN {X 0,Y 281.014,Z 542.301,A -85,B 0,C 180,E1 -17390.685,E2 -17390.685} C_VEL
LIN {X 0,Y 282.16,Z 533.158,A -85,B 0,C 180,E1 -17391.937,E2 -17391.937} C_VEL
LIN {X 0,Y 281.544,Z 520.744,A -85,B 0,C 180,E1 -17393.539,E2 -17393.539} C_VEL
LIN {X 0,Y 280.46,Z 506.095,A -85,B 0,C 180,E1 -17395.113,E2 -17395.113} C_VEL
LIN {X 0,Y 279.43,Z 492.255,A -85,B 0,C 180,E1 -17396.311,E2 -17396.311} C_VEL
LIN {X 0,Y 278.208,Z 476.748,A -85,B 0,C 180,E1 -17397.352,E2 -17397.352} C_VEL
LIN {X 0,Y 277.736,Z 469.877,A -85,B 0,C 180,E1 -17397.755,E2 -17397.755} C_VEL
LIN {X 0,Y 279.177,Z 458.599,A -85,B 0,C 180,E1 -17402.766,E2 -17402.766} C_VEL
LIN {X 0,Y 280.642,Z 449.258,A -85,B 0,C 180,E1 -17406.941,E2 -17406.941} C_VEL
LIN {X 0,Y 281.988,Z 441.66,A -85,B 0,C 180,E1 -17410.388,E2 -17410.388} C_VEL
LIN {X 0,Y 282.111,Z 438.982,A -85,B 0,C 180,E1 -17411.638,E2 -17411.638} C_VEL
LIN {X 0,Y 280.561,Z 431.204,A -85,B 0,C 180,E1 -17415.461,E2 -17415.461} C_VEL
LIN {X 0,Y 279.129,Z 424.112,A -85,B 0,C 180,E1 -17419.108,E2 -17419.108} C_VEL
LIN {X 0,Y 277.857,Z 417.561,A -85,B 0,C 180,E1 -17422.624,E2 -17422.624} C_VEL
LIN {X 0,Y 277.299,Z 414.569,A -85,B 0,C 180,E1 -17424.344,E2 -17424.344} C_VEL
LIN {X 0,Y 277.236,Z 414.575,A -85,B 0,C 180,E1 -17427.836,E2 -17427.836} C_VEL
LIN {X 0,Y 277.282,Z 414.569,A -85,B 0,C 180,E1 -17431.212,E2 -17431.212} C_VEL
LIN {X 0,Y 277.306,Z 414.565,A -85,B 0,C 180,E1 -17434.479,E2 -17434.479} C_VEL
LIN {X 0,Y 277.275,Z 414.57,A -85,B 0,C 180,E1 -17437.654,E2 -17437.654} C_VEL
LIN {X 0,Y 277.335,Z 414.561,A -85,B 0,C 180,E1 -17440.766,E2 -17440.766} C_VEL
LIN {X 0,Y 277.425,Z 414.551,A -85,B 0,C 180,E1 -17445.326,E2 -17445.326} C_VEL
LIN {X 0,Y 277.497,Z 414.537,A -85,B 0,C 180,E1 -17449.789,E2 -17449.789} C_VEL
LIN {X 0,Y 277.643,Z 414.526,A -85,B 0,C 180,E1 -17452.729,E2 -17452.729} C_VEL
LIN {X 0,Y 277.816,Z 414.504,A -85,B 0,C 180,E1 -17458.551,E2 -17458.551} C_VEL
LIN {X 0,Y 277.816,Z 414.501,A -85,B 0,C 180,E1 -17461.45,E2 -17461.45} C_VEL
LIN {X 0,Y 277.644,Z 414.512,A -85,B 0,C 180,E1 -17467.272,E2 -17467.272} C_VEL
LIN {X 0,Y 277.498,Z 414.528,A -85,B 0,C 180,E1 -17470.212,E2 -17470.212} C_VEL
LIN {X 0,Y 277.426,Z 414.555,A -85,B 0,C 180,E1 -17474.675,E2 -17474.675} C_VEL
LIN {X 0,Y 277.337,Z 414.563,A -85,B 0,C 180,E1 -17479.235,E2 -17479.235} C_VEL
LIN {X 0,Y 277.311,Z 414.565,A -85,B 0,C 180,E1 -17484.172,E2 -17484.172} C_VEL
LIN {X 0,Y 277.318,Z 414.558,A -85,B 0,C 180,E1 -17487.507,E2 -17487.507} C_VEL
LIN {X 0,Y 277.265,Z 414.556,A -85,B 0,C 180,E1 -17490.483,E2 -17490.483} C_VEL
